Fanuc TP program (LS listing): hs0301h80_2.ls

/PROG  hs0301h80_2
/ATTR
COMMENT	= "19-03-01 11:47:14";
PROG_SIZE	= 0;
DEFAULT_GROUP	= 1, *, *, *, *;
/APPL
    ARC Welding Equipment: 1, *, *, *, *;
/MN
   1:  CALL HOME_ALL;
   1:  UFRAME_NUM = 1;
   1:  UTOOL_NUM = 3;
   1:  COL GUARD ADJUST 150;
   1:  PR[91] = PR[90];
   1:  PR[91,1] = PR[90,1] + -0.666;
   1:  PR[91,2] = PR[90,2] + 15.331;
   1:  PR[91,3] = PR[90,3] + 35.075;
   1:  PR[92] = PR[91];
   1:  PR[92,3] = PR[92,3] + 50;
   1:J PR[92] 10% FINE;
   1:L PR[91] R[100]mm/sec CNT100;
   1:  CALL LASER_DRAHT_START;
   1:  PR[91,1] = PR[90,1] + -0.927;
   1:  PR[91,2] = PR[90,2] + 15.462;
   1:L PR[91] R[100]mm/sec CNT100;
   1:  PR[91,1] = PR[90,1] + -1.615;
   1:  PR[91,2] = PR[90,2] + 15.721;
   1:L PR[91] R[100]mm/sec CNT100;
   1:  PR[91,1] = PR[90,1] + -2.354;
   1:  PR[91,2] = PR[90,2] + 16.306;
   1:L PR[91] R[100]mm/sec CNT100;
   1:  PR[91,1] = PR[90,1] + -3.858;
   1:  PR[91,2] = PR[90,2] + 17.303;
   1:L PR[91] R[100]mm/sec CNT100;
   1:  PR[91,1] = PR[90,1] + -4.809;
   1:  PR[91,2] = PR[90,2] + 17.719;
   1:L PR[91] R[100]mm/sec CNT100;
   1:  PR[91,1] = PR[90,1] + -8.585;
   1:  PR[91,2] = PR[90,2] + 19.301;
   1:L PR[91] R[100]mm/sec CNT100;
   1:  PR[91,1] = PR[90,1] + -9.692;
   1:  PR[91,2] = PR[90,2] + 19.587;
   1:L PR[91] R[100]mm/sec CNT100;
   1:  PR[91,1] = PR[90,1] + -11.119;
   1:  PR[91,2] = PR[90,2] + 19.736;
   1:L PR[91] R[100]mm/sec CNT100;
   1:  PR[91,1] = PR[90,1] + -14.708;
   1:  PR[91,2] = PR[90,2] + 20.226;
   1:L PR[91] R[100]mm/sec CNT100;
   1:  PR[91,1] = PR[90,1] + -16.221;
   1:  PR[91,2] = PR[90,2] + 20.146;
   1:L PR[91] R[100]mm/sec CNT100;
   1:  PR[91,1] = PR[90,1] + -19.349;
   1:  PR[91,2] = PR[90,2] + 19.776;
   1:L PR[91] R[100]mm/sec CNT100;
   1:  PR[91,1] = PR[90,1] + -20.989;
   1:  PR[91,2] = PR[90,2] + 19.436;
   1:L PR[91] R[100]mm/sec CNT100;
   1:  PR[91,1] = PR[90,1] + -22.810;
   1:  PR[91,2] = PR[90,2] + 18.760;
   1:L PR[91] R[100]mm/sec CNT100;
   1:  PR[91,1] = PR[90,1] + -25.231;
   1:  PR[91,2] = PR[90,2] + 17.813;
   1:L PR[91] R[100]mm/sec CNT100;
   1:  PR[91,1] = PR[90,1] + -26.962;
   1:  PR[91,2] = PR[90,2] + 16.843;
   1:L PR[91] R[100]mm/sec CNT100;
   1:  PR[91,1] = PR[90,1] + -28.774;
   1:  PR[91,2] = PR[90,2] + 15.433;
   1:L PR[91] R[100]mm/sec CNT100;
   1:  PR[91,1] = PR[90,1] + -30.430;
   1:  PR[91,2] = PR[90,2] + 14.227;
   1:L PR[91] R[100]mm/sec CNT100;
   1:  PR[91,1] = PR[90,1] + -31.950;
   1:  PR[91,2] = PR[90,2] + 12.586;
   1:L PR[91] R[100]mm/sec CNT100;
   1:  PR[91,1] = PR[90,1] + -33.021;
   1:  PR[91,2] = PR[90,2] + 11.255;
   1:L PR[91] R[100]mm/sec CNT100;
   1:  PR[91,1] = PR[90,1] + -34.310;
   1:  PR[91,2] = PR[90,2] + 9.296;
   1:L PR[91] R[100]mm/sec CNT100;
   1:  PR[91,1] = PR[90,1] + -35.922;
   1:  PR[91,2] = PR[90,2] + 5.672;
   1:L PR[91] R[100]mm/sec CNT100;
   1:  PR[91,1] = PR[90,1] + -36.506;
   1:  PR[91,2] = PR[90,2] + 3.415;
   1:L PR[91] R[100]mm/sec CNT100;
   1:  PR[91,1] = PR[90,1] + -36.709;
   1:  PR[91,2] = PR[90,2] + 0.880;
   1:L PR[91] R[100]mm/sec CNT100;
   1:  PR[91,1] = PR[90,1] + -36.880;
   1:  PR[91,2] = PR[90,2] + -0.354;
   1:L PR[91] R[100]mm/sec CNT100;
   1:  PR[91,1] = PR[90,1] + -36.688;
   1:  PR[91,2] = PR[90,2] + -2.767;
   1:L PR[91] R[100]mm/sec CNT100;
   1:  PR[91,1] = PR[90,1] + -36.517;
   1:  PR[91,2] = PR[90,2] + -3.999;
   1:L PR[91] R[100]mm/sec CNT100;
   1:  PR[91,1] = PR[90,1] + -35.922;
   1:  PR[91,2] = PR[90,2] + -6.296;
   1:L PR[91] R[100]mm/sec CNT100;
   1:  PR[91,1] = PR[90,1] + -34.892;
   1:  PR[91,2] = PR[90,2] + -8.592;
   1:L PR[91] R[100]mm/sec CNT100;
   1:  PR[91,1] = PR[90,1] + -34.306;
   1:  PR[91,2] = PR[90,2] + -9.927;
   1:L PR[91] R[100]mm/sec CNT100;
   1:  PR[91,1] = PR[90,1] + -33.019;
   1:  PR[91,2] = PR[90,2] + -11.883;
   1:L PR[91] R[100]mm/sec CNT100;
   1:  PR[91,1] = PR[90,1] + -31.945;
   1:  PR[91,2] = PR[90,2] + -13.214;
   1:L PR[91] R[100]mm/sec CNT100;
   1:  PR[91,1] = PR[90,1] + -30.408;
   1:  PR[91,2] = PR[90,2] + -14.874;
   1:L PR[91] R[100]mm/sec CNT100;
   1:  PR[91,1] = PR[90,1] + -28.736;
   1:  PR[91,2] = PR[90,2] + -16.183;
   1:L PR[91] R[100]mm/sec CNT100;
   1:  PR[91,1] = PR[90,1] + -26.973;
   1:  PR[91,2] = PR[90,2] + -17.461;
   1:L PR[91] R[100]mm/sec CNT100;
   1:  PR[91,1] = PR[90,1] + -25.232;
   1:  PR[91,2] = PR[90,2] + -18.437;
   1:L PR[91] R[100]mm/sec CNT100;
   1:  PR[91,1] = PR[90,1] + -23.475;
   1:  PR[91,2] = PR[90,2] + -19.085;
   1:L PR[91] R[100]mm/sec CNT100;
   1:  PR[91,1] = PR[90,1] + -20.959;
   1:  PR[91,2] = PR[90,2] + -20.067;
   1:L PR[91] R[100]mm/sec CNT100;
   1:  PR[91,1] = PR[90,1] + -19.331;
   1:  PR[91,2] = PR[90,2] + -20.404;
   1:L PR[91] R[100]mm/sec CNT100;
   1:  PR[91,1] = PR[90,1] + -16.196;
   1:  PR[91,2] = PR[90,2] + -20.770;
   1:L PR[91] R[100]mm/sec CNT100;
   1:  PR[91,1] = PR[90,1] + -14.656;
   1:  PR[91,2] = PR[90,2] + -20.851;
   1:L PR[91] R[100]mm/sec CNT100;
   1:  PR[91,1] = PR[90,1] + -13.288;
   1:  PR[91,2] = PR[90,2] + -20.713;
   1:L PR[91] R[100]mm/sec CNT100;
   1:  PR[91,1] = PR[90,1] + -9.682;
   1:  PR[91,2] = PR[90,2] + -20.208;
   1:L PR[91] R[100]mm/sec CNT100;
   1:  PR[91,1] = PR[90,1] + -8.557;
   1:  PR[91,2] = PR[90,2] + -19.917;
   1:L PR[91] R[100]mm/sec CNT100;
   1:  PR[91,1] = PR[90,1] + -3.731;
   1:  PR[91,2] = PR[90,2] + -17.847;
   1:L PR[91] R[100]mm/sec CNT100;
   1:  PR[91,1] = PR[90,1] + -3.017;
   1:  PR[91,2] = PR[90,2] + -17.391;
   1:L PR[91] R[100]mm/sec CNT100;
   1:  PR[91,1] = PR[90,1] + -1.910;
   1:  PR[91,2] = PR[90,2] + -16.593;
   1:L PR[91] R[100]mm/sec CNT100;
   1:  PR[91,1] = PR[90,1] + -1.659;
   1:  PR[91,2] = PR[90,2] + -16.373;
   1:L PR[91] R[100]mm/sec CNT100;
   1:  PR[91,1] = PR[90,1] + 0.008;
   1:  PR[91,2] = PR[90,2] + -15.711;
   1:L PR[91] R[100]mm/sec CNT100;
   1:  PR[91,1] = PR[90,1] + 0.793;
   1:  PR[91,2] = PR[90,2] + -16.025;
   1:L PR[91] R[100]mm/sec CNT100;
   1:  PR[91,1] = PR[90,1] + 1.694;
   1:  PR[91,2] = PR[90,2] + -16.187;
   1:L PR[91] R[100]mm/sec CNT100;
   1:  PR[91,1] = PR[90,1] + 2.030;
   1:  PR[91,2] = PR[90,2] + -16.568;
   1:L PR[91] R[100]mm/sec CNT100;
   1:  PR[91,1] = PR[90,1] + 2.042;
   1:  PR[91,2] = PR[90,2] + -16.578;
   1:L PR[91] R[100]mm/sec CNT100;
   1:  PR[91,1] = PR[90,1] + 2.791;
   1:  PR[91,2] = PR[90,2] + -17.107;
   1:L PR[91] R[100]mm/sec CNT100;
   1:  PR[91,1] = PR[90,1] + 3.899;
   1:  PR[91,2] = PR[90,2] + -17.854;
   1:L PR[91] R[100]mm/sec CNT100;
   1:  PR[91,1] = PR[90,1] + 8.708;
   1:  PR[91,2] = PR[90,2] + -19.914;
   1:L PR[91] R[100]mm/sec CNT100;
   1:  PR[91,1] = PR[90,1] + 9.812;
   1:  PR[91,2] = PR[90,2] + -20.200;
   1:L PR[91] R[100]mm/sec CNT100;
   1:  PR[91,1] = PR[90,1] + 11.237;
   1:  PR[91,2] = PR[90,2] + -20.349;
   1:L PR[91] R[100]mm/sec CNT100;
   1:  PR[91,1] = PR[90,1] + 14.834;
   1:  PR[91,2] = PR[90,2] + -20.850;
   1:L PR[91] R[100]mm/sec CNT100;
   1:  PR[91,1] = PR[90,1] + 16.338;
   1:  PR[91,2] = PR[90,2] + -20.771;
   1:L PR[91] R[100]mm/sec CNT100;
   1:  PR[91,1] = PR[90,1] + 19.474;
   1:  PR[91,2] = PR[90,2] + -20.406;
   1:L PR[91] R[100]mm/sec CNT100;
   1:  PR[91,1] = PR[90,1] + 21.112;
   1:  PR[91,2] = PR[90,2] + -20.067;
   1:L PR[91] R[100]mm/sec CNT100;
   1:  PR[91,1] = PR[90,1] + 22.936;
   1:  PR[91,2] = PR[90,2] + -19.393;
   1:L PR[91] R[100]mm/sec CNT100;
   1:  PR[91,1] = PR[90,1] + 25.366;
   1:  PR[91,2] = PR[90,2] + -18.448;
   1:L PR[91] R[100]mm/sec CNT100;
   1:  PR[91,1] = PR[90,1] + 27.089;
   1:  PR[91,2] = PR[90,2] + -17.488;
   1:L PR[91] R[100]mm/sec CNT100;
   1:  PR[91,1] = PR[90,1] + 28.887;
   1:  PR[91,2] = PR[90,2] + -16.095;
   1:L PR[91] R[100]mm/sec CNT100;
   1:  PR[91,1] = PR[90,1] + 30.549;
   1:  PR[91,2] = PR[90,2] + -14.888;
   1:L PR[91] R[100]mm/sec CNT100;
   1:  PR[91,1] = PR[90,1] + 32.072;
   1:  PR[91,2] = PR[90,2] + -13.246;
   1:L PR[91] R[100]mm/sec CNT100;
   1:  PR[91,1] = PR[90,1] + 33.148;
   1:  PR[91,2] = PR[90,2] + -11.909;
   1:L PR[91] R[100]mm/sec CNT100;
   1:  PR[91,1] = PR[90,1] + 34.457;
   1:  PR[91,2] = PR[90,2] + -9.931;
   1:L PR[91] R[100]mm/sec CNT100;
   1:  PR[91,1] = PR[90,1] + 35.518;
   1:  PR[91,2] = PR[90,2] + -7.595;
   1:L PR[91] R[100]mm/sec CNT100;
   1:  PR[91,1] = PR[90,1] + 36.065;
   1:  PR[91,2] = PR[90,2] + -6.353;
   1:L PR[91] R[100]mm/sec CNT100;
   1:  PR[91,1] = PR[90,1] + 36.652;
   1:  PR[91,2] = PR[90,2] + -4.119;
   1:L PR[91] R[100]mm/sec CNT100;
   1:  PR[91,1] = PR[90,1] + 36.866;
   1:  PR[91,2] = PR[90,2] + -1.508;
   1:L PR[91] R[100]mm/sec CNT100;
   1:  PR[91,1] = PR[90,1] + 37.037;
   1:  PR[91,2] = PR[90,2] + -0.271;
   1:L PR[91] R[100]mm/sec CNT100;
   1:  PR[91,1] = PR[90,1] + 36.834;
   1:  PR[91,2] = PR[90,2] + 2.220;
   1:L PR[91] R[100]mm/sec CNT100;
   1:  PR[91,1] = PR[90,1] + 36.662;
   1:  PR[91,2] = PR[90,2] + 3.454;
   1:L PR[91] R[100]mm/sec CNT100;
   1:  PR[91,1] = PR[90,1] + 36.068;
   1:  PR[91,2] = PR[90,2] + 5.720;
   1:L PR[91] R[100]mm/sec CNT100;
   1:  PR[91,1] = PR[90,1] + 35.039;
   1:  PR[91,2] = PR[90,2] + 7.981;
   1:L PR[91] R[100]mm/sec CNT100;
   1:  PR[91,1] = PR[90,1] + 34.455;
   1:  PR[91,2] = PR[90,2] + 9.310;
   1:L PR[91] R[100]mm/sec CNT100;
   1:  PR[91,1] = PR[90,1] + 33.150;
   1:  PR[91,2] = PR[90,2] + 11.281;
   1:L PR[91] R[100]mm/sec CNT100;
   1:  PR[91,1] = PR[90,1] + 32.076;
   1:  PR[91,2] = PR[90,2] + 12.617;
   1:L PR[91] R[100]mm/sec CNT100;
   1:  PR[91,1] = PR[90,1] + 30.537;
   1:  PR[91,2] = PR[90,2] + 14.277;
   1:L PR[91] R[100]mm/sec CNT100;
   1:  PR[91,1] = PR[90,1] + 28.879;
   1:  PR[91,2] = PR[90,2] + 15.569;
   1:L PR[91] R[100]mm/sec CNT100;
   1:  PR[91,1] = PR[90,1] + 27.119;
   1:  PR[91,2] = PR[90,2] + 16.848;
   1:L PR[91] R[100]mm/sec CNT100;
   1:  PR[91,1] = PR[90,1] + 25.389;
   1:  PR[91,2] = PR[90,2] + 17.812;
   1:L PR[91] R[100]mm/sec CNT100;
   1:  PR[91,1] = PR[90,1] + 23.629;
   1:  PR[91,2] = PR[90,2] + 18.459;
   1:L PR[91] R[100]mm/sec CNT100;
   1:  PR[91,1] = PR[90,1] + 21.116;
   1:  PR[91,2] = PR[90,2] + 19.442;
   1:L PR[91] R[100]mm/sec CNT100;
   1:  PR[91,1] = PR[90,1] + 19.492;
   1:  PR[91,2] = PR[90,2] + 19.778;
   1:L PR[91] R[100]mm/sec CNT100;
   1:  PR[91,1] = PR[90,1] + 16.363;
   1:  PR[91,2] = PR[90,2] + 20.148;
   1:L PR[91] R[100]mm/sec CNT100;
   1:  PR[91,1] = PR[90,1] + 14.834;
   1:  PR[91,2] = PR[90,2] + 20.227;
   1:L PR[91] R[100]mm/sec CNT100;
   1:  PR[91,1] = PR[90,1] + 13.468;
   1:  PR[91,2] = PR[90,2] + 20.089;
   1:L PR[91] R[100]mm/sec CNT100;
   1:  PR[91,1] = PR[90,1] + 9.868;
   1:  PR[91,2] = PR[90,2] + 19.591;
   1:L PR[91] R[100]mm/sec CNT100;
   1:  PR[91,1] = PR[90,1] + 8.747;
   1:  PR[91,2] = PR[90,2] + 19.300;
   1:L PR[91] R[100]mm/sec CNT100;
   1:  PR[91,1] = PR[90,1] + 7.722;
   1:  PR[91,2] = PR[90,2] + 18.852;
   1:L PR[91] R[100]mm/sec CNT100;
   1:  PR[91,1] = PR[90,1] + 3.989;
   1:  PR[91,2] = PR[90,2] + 17.292;
   1:L PR[91] R[100]mm/sec CNT100;
   1:  PR[91,1] = PR[90,1] + 3.235;
   1:  PR[91,2] = PR[90,2] + 16.810;
   1:L PR[91] R[100]mm/sec CNT100;
   1:  PR[91,1] = PR[90,1] + 2.521;
   1:  PR[91,2] = PR[90,2] + 16.318;
   1:L PR[91] R[100]mm/sec CNT100;
   1:  PR[91,1] = PR[90,1] + 2.001;
   1:  PR[91,2] = PR[90,2] + 15.906;
   1:L PR[91] R[100]mm/sec CNT100;
   1:  PR[91,1] = PR[90,1] + 1.619;
   1:  PR[91,2] = PR[90,2] + 15.536;
   1:L PR[91] R[100]mm/sec CNT100;
   1:  PR[91,1] = PR[90,1] + 0.760;
   1:  PR[91,2] = PR[90,2] + 15.389;
   1:L PR[91] R[100]mm/sec CNT100;
   1:  PR[91,1] = PR[90,1] + 0.087;
   1:  PR[91,2] = PR[90,2] + 15.117;
   1:L PR[91] R[100]mm/sec CNT100;
   1:  PR[91] = PR[90];
   1:  PR[91,1] = PR[90,1] + -0.722;
   1:  PR[91,2] = PR[90,2] + 15.588;
   1:  PR[91,3] = PR[90,3] + 35.685;
   1:L PR[91] R[100]mm/sec CNT100;
   1:  PR[91,1] = PR[90,1] + -1.091;
   1:  PR[91,2] = PR[90,2] + 15.774;
   1:L PR[91] R[100]mm/sec CNT100;
   1:  PR[91,1] = PR[90,1] + -1.597;
   1:  PR[91,2] = PR[90,2] + 15.965;
   1:L PR[91] R[100]mm/sec CNT100;
   1:  PR[91,1] = PR[90,1] + -2.135;
   1:  PR[91,2] = PR[90,2] + 16.391;
   1:L PR[91] R[100]mm/sec CNT100;
   1:  PR[91,1] = PR[90,1] + -3.572;
   1:  PR[91,2] = PR[90,2] + 17.346;
   1:L PR[91] R[100]mm/sec CNT100;
   1:  PR[91,1] = PR[90,1] + -4.394;
   1:  PR[91,2] = PR[90,2] + 17.706;
   1:L PR[91] R[100]mm/sec CNT100;
   1:  PR[91,1] = PR[90,1] + -8.389;
   1:  PR[91,2] = PR[90,2] + 19.380;
   1:L PR[91] R[100]mm/sec CNT100;
   1:  PR[91,1] = PR[90,1] + -9.367;
   1:  PR[91,2] = PR[90,2] + 19.633;
   1:L PR[91] R[100]mm/sec CNT100;
   1:  PR[91,1] = PR[90,1] + -10.645;
   1:  PR[91,2] = PR[90,2] + 19.766;
   1:L PR[91] R[100]mm/sec CNT100;
   1:  PR[91,1] = PR[90,1] + -14.484;
   1:  PR[91,2] = PR[90,2] + 20.290;
   1:L PR[91] R[100]mm/sec CNT100;
   1:  PR[91,1] = PR[90,1] + -15.854;
   1:  PR[91,2] = PR[90,2] + 20.217;
   1:L PR[91] R[100]mm/sec CNT100;
   1:  PR[91,1] = PR[90,1] + -19.224;
   1:  PR[91,2] = PR[90,2] + 19.819;
   1:L PR[91] R[100]mm/sec CNT100;
   1:  PR[91,1] = PR[90,1] + -20.730;
   1:  PR[91,2] = PR[90,2] + 19.506;
   1:L PR[91] R[100]mm/sec CNT100;
   1:  PR[91,1] = PR[90,1] + -22.409;
   1:  PR[91,2] = PR[90,2] + 18.883;
   1:L PR[91] R[100]mm/sec CNT100;
   1:  PR[91,1] = PR[90,1] + -25.070;
   1:  PR[91,2] = PR[90,2] + 17.843;
   1:L PR[91] R[100]mm/sec CNT100;
   1:  PR[91,1] = PR[90,1] + -26.674;
   1:  PR[91,2] = PR[90,2] + 16.944;
   1:L PR[91] R[100]mm/sec CNT100;
   1:  PR[91,1] = PR[90,1] + -28.363;
   1:  PR[91,2] = PR[90,2] + 15.630;
   1:L PR[91] R[100]mm/sec CNT100;
   1:  PR[91,1] = PR[90,1] + -30.234;
   1:  PR[91,2] = PR[90,2] + 14.267;
   1:L PR[91] R[100]mm/sec CNT100;
   1:  PR[91,1] = PR[90,1] + -31.654;
   1:  PR[91,2] = PR[90,2] + 12.733;
   1:L PR[91] R[100]mm/sec CNT100;
   1:  PR[91,1] = PR[90,1] + -32.885;
   1:  PR[91,2] = PR[90,2] + 11.204;
   1:L PR[91] R[100]mm/sec CNT100;
   1:  PR[91,1] = PR[90,1] + -34.095;
   1:  PR[91,2] = PR[90,2] + 9.366;
   1:L PR[91] R[100]mm/sec CNT100;
   1:  PR[91,1] = PR[90,1] + -35.747;
   1:  PR[91,2] = PR[90,2] + 5.647;
   1:L PR[91] R[100]mm/sec CNT100;
   1:  PR[91,1] = PR[90,1] + -36.296;
   1:  PR[91,2] = PR[90,2] + 3.526;
   1:L PR[91] R[100]mm/sec CNT100;
   1:  PR[91,1] = PR[90,1] + -36.488;
   1:  PR[91,2] = PR[90,2] + 1.135;
   1:L PR[91] R[100]mm/sec CNT100;
   1:  PR[91,1] = PR[90,1] + -36.694;
   1:  PR[91,2] = PR[90,2] + -0.354;
   1:L PR[91] R[100]mm/sec CNT100;
   1:  PR[91,1] = PR[90,1] + -36.513;
   1:  PR[91,2] = PR[90,2] + -2.628;
   1:L PR[91] R[100]mm/sec CNT100;
   1:  PR[91,1] = PR[90,1] + -36.306;
   1:  PR[91,2] = PR[90,2] + -4.111;
   1:L PR[91] R[100]mm/sec CNT100;
   1:  PR[91,1] = PR[90,1] + -35.747;
   1:  PR[91,2] = PR[90,2] + -6.271;
   1:L PR[91] R[100]mm/sec CNT100;
   1:  PR[91,1] = PR[90,1] + -34.776;
   1:  PR[91,2] = PR[90,2] + -8.435;
   1:L PR[91] R[100]mm/sec CNT100;
   1:  PR[91,1] = PR[90,1] + -34.091;
   1:  PR[91,2] = PR[90,2] + -9.996;
   1:L PR[91] R[100]mm/sec CNT100;
   1:  PR[91,1] = PR[90,1] + -32.883;
   1:  PR[91,2] = PR[90,2] + -11.832;
   1:L PR[91] R[100]mm/sec CNT100;
   1:  PR[91,1] = PR[90,1] + -31.648;
   1:  PR[91,2] = PR[90,2] + -13.363;
   1:L PR[91] R[100]mm/sec CNT100;
   1:  PR[91,1] = PR[90,1] + -30.211;
   1:  PR[91,2] = PR[90,2] + -14.915;
   1:L PR[91] R[100]mm/sec CNT100;
   1:  PR[91,1] = PR[90,1] + -28.647;
   1:  PR[91,2] = PR[90,2] + -16.139;
   1:L PR[91] R[100]mm/sec CNT100;
   1:  PR[91,1] = PR[90,1] + -26.684;
   1:  PR[91,2] = PR[90,2] + -17.563;
   1:L PR[91] R[100]mm/sec CNT100;
   1:  PR[91,1] = PR[90,1] + -25.069;
   1:  PR[91,2] = PR[90,2] + -18.467;
   1:L PR[91] R[100]mm/sec CNT100;
   1:  PR[91,1] = PR[90,1] + -23.435;
   1:  PR[91,2] = PR[90,2] + -19.071;
   1:L PR[91] R[100]mm/sec CNT100;
   1:  PR[91,1] = PR[90,1] + -20.699;
   1:  PR[91,2] = PR[90,2] + -20.138;
   1:L PR[91] R[100]mm/sec CNT100;
   1:  PR[91,1] = PR[90,1] + -19.205;
   1:  PR[91,2] = PR[90,2] + -20.448;
   1:L PR[91] R[100]mm/sec CNT100;
   1:  PR[91,1] = PR[90,1] + -15.826;
   1:  PR[91,2] = PR[90,2] + -20.841;
   1:L PR[91] R[100]mm/sec CNT100;
   1:  PR[91,1] = PR[90,1] + -14.430;
   1:  PR[91,2] = PR[90,2] + -20.915;
   1:L PR[91] R[100]mm/sec CNT100;
   1:  PR[91,1] = PR[90,1] + -13.190;
   1:  PR[91,2] = PR[90,2] + -20.790;
   1:L PR[91] R[100]mm/sec CNT100;
   1:  PR[91,1] = PR[90,1] + -9.355;
   1:  PR[91,2] = PR[90,2] + -20.253;
   1:L PR[91] R[100]mm/sec CNT100;
   1:  PR[91,1] = PR[90,1] + -8.359;
   1:  PR[91,2] = PR[90,2] + -19.996;
   1:L PR[91] R[100]mm/sec CNT100;
   1:  PR[91,1] = PR[90,1] + -3.437;
   1:  PR[91,2] = PR[90,2] + -17.886;
   1:L PR[91] R[100]mm/sec CNT100;
   1:  PR[91,1] = PR[90,1] + -2.832;
   1:  PR[91,2] = PR[90,2] + -17.500;
   1:L PR[91] R[100]mm/sec CNT100;
   1:  PR[91,1] = PR[90,1] + -1.582;
   1:  PR[91,2] = PR[90,2] + -16.598;
   1:L PR[91] R[100]mm/sec CNT100;
   1:  PR[91,1] = PR[90,1] + 0.021;
   1:  PR[91,2] = PR[90,2] + -15.944;
   1:L PR[91] R[100]mm/sec CNT100;
   1:  PR[91,1] = PR[90,1] + 1.017;
   1:  PR[91,2] = PR[90,2] + -16.343;
   1:L PR[91] R[100]mm/sec CNT100;
   1:  PR[91,1] = PR[90,1] + 1.715;
   1:  PR[91,2] = PR[90,2] + -16.468;
   1:L PR[91] R[100]mm/sec CNT100;
   1:  PR[91,1] = PR[90,1] + 2.003;
   1:  PR[91,2] = PR[90,2] + -16.795;
   1:L PR[91] R[100]mm/sec CNT100;
   1:  PR[91,1] = PR[90,1] + 2.436;
   1:  PR[91,2] = PR[90,2] + -17.104;
   1:L PR[91] R[100]mm/sec CNT100;
   1:  PR[91,1] = PR[90,1] + 3.606;
   1:  PR[91,2] = PR[90,2] + -17.893;
   1:L PR[91] R[100]mm/sec CNT100;
   1:  PR[91,1] = PR[90,1] + 8.511;
   1:  PR[91,2] = PR[90,2] + -19.992;
   1:L PR[91] R[100]mm/sec CNT100;
   1:  PR[91,1] = PR[90,1] + 9.485;
   1:  PR[91,2] = PR[90,2] + -20.245;
   1:L PR[91] R[100]mm/sec CNT100;
   1:  PR[91,1] = PR[90,1] + 10.761;
   1:  PR[91,2] = PR[90,2] + -20.379;
   1:L PR[91] R[100]mm/sec CNT100;
   1:  PR[91,1] = PR[90,1] + 14.609;
   1:  PR[91,2] = PR[90,2] + -20.914;
   1:L PR[91] R[100]mm/sec CNT100;
   1:  PR[91,1] = PR[90,1] + 15.970;
   1:  PR[91,2] = PR[90,2] + -20.843;
   1:L PR[91] R[100]mm/sec CNT100;
   1:  PR[91,1] = PR[90,1] + 19.349;
   1:  PR[91,2] = PR[90,2] + -20.449;
   1:L PR[91] R[100]mm/sec CNT100;
   1:  PR[91,1] = PR[90,1] + 20.853;
   1:  PR[91,2] = PR[90,2] + -20.138;
   1:L PR[91] R[100]mm/sec CNT100;
   1:  PR[91,1] = PR[90,1] + 22.535;
   1:  PR[91,2] = PR[90,2] + -19.517;
   1:L PR[91] R[100]mm/sec CNT100;
   1:  PR[91,1] = PR[90,1] + 25.204;
   1:  PR[91,2] = PR[90,2] + -18.479;
   1:L PR[91] R[100]mm/sec CNT100;
   1:  PR[91,1] = PR[90,1] + 26.802;
   1:  PR[91,2] = PR[90,2] + -17.589;
   1:L PR[91] R[100]mm/sec CNT100;
   1:  PR[91,1] = PR[90,1] + 28.476;
   1:  PR[91,2] = PR[90,2] + -16.291;
   1:L PR[91] R[100]mm/sec CNT100;
   1:  PR[91,1] = PR[90,1] + 30.354;
   1:  PR[91,2] = PR[90,2] + -14.927;
   1:L PR[91] R[100]mm/sec CNT100;
   1:  PR[91,1] = PR[90,1] + 31.777;
   1:  PR[91,2] = PR[90,2] + -13.392;
   1:L PR[91] R[100]mm/sec CNT100;
   1:  PR[91,1] = PR[90,1] + 33.014;
   1:  PR[91,2] = PR[90,2] + -11.856;
   1:L PR[91] R[100]mm/sec CNT100;
   1:  PR[91,1] = PR[90,1] + 34.242;
   1:  PR[91,2] = PR[90,2] + -10.000;
   1:L PR[91] R[100]mm/sec CNT100;
   1:  PR[91,1] = PR[90,1] + 35.240;
   1:  PR[91,2] = PR[90,2] + -7.803;
   1:L PR[91] R[100]mm/sec CNT100;
   1:  PR[91,1] = PR[90,1] + 35.891;
   1:  PR[91,2] = PR[90,2] + -6.326;
   1:L PR[91] R[100]mm/sec CNT100;
   1:  PR[91,1] = PR[90,1] + 36.442;
   1:  PR[91,2] = PR[90,2] + -4.227;
   1:L PR[91] R[100]mm/sec CNT100;
   1:  PR[91,1] = PR[90,1] + 36.644;
   1:  PR[91,2] = PR[90,2] + -1.764;
   1:L PR[91] R[100]mm/sec CNT100;
   1:  PR[91,1] = PR[90,1] + 36.851;
   1:  PR[91,2] = PR[90,2] + -0.271;
   1:L PR[91] R[100]mm/sec CNT100;
   1:  PR[91,1] = PR[90,1] + 36.659;
   1:  PR[91,2] = PR[90,2] + 2.076;
   1:L PR[91] R[100]mm/sec CNT100;
   1:  PR[91,1] = PR[90,1] + 36.453;
   1:  PR[91,2] = PR[90,2] + 3.562;
   1:L PR[91] R[100]mm/sec CNT100;
   1:  PR[91,1] = PR[90,1] + 35.894;
   1:  PR[91,2] = PR[90,2] + 5.692;
   1:L PR[91] R[100]mm/sec CNT100;
   1:  PR[91,1] = PR[90,1] + 34.924;
   1:  PR[91,2] = PR[90,2] + 7.824;
   1:L PR[91] R[100]mm/sec CNT100;
   1:  PR[91,1] = PR[90,1] + 34.240;
   1:  PR[91,2] = PR[90,2] + 9.379;
   1:L PR[91] R[100]mm/sec CNT100;
   1:  PR[91,1] = PR[90,1] + 33.016;
   1:  PR[91,2] = PR[90,2] + 11.228;
   1:L PR[91] R[100]mm/sec CNT100;
   1:  PR[91,1] = PR[90,1] + 31.782;
   1:  PR[91,2] = PR[90,2] + 12.763;
   1:L PR[91] R[100]mm/sec CNT100;
   1:  PR[91,1] = PR[90,1] + 30.343;
   1:  PR[91,2] = PR[90,2] + 14.315;
   1:L PR[91] R[100]mm/sec CNT100;
   1:  PR[91,1] = PR[90,1] + 28.792;
   1:  PR[91,2] = PR[90,2] + 15.524;
   1:L PR[91] R[100]mm/sec CNT100;
   1:  PR[91,1] = PR[90,1] + 26.833;
   1:  PR[91,2] = PR[90,2] + 16.947;
   1:L PR[91] R[100]mm/sec CNT100;
   1:  PR[91,1] = PR[90,1] + 25.228;
   1:  PR[91,2] = PR[90,2] + 17.841;
   1:L PR[91] R[100]mm/sec CNT100;
   1:  PR[91,1] = PR[90,1] + 23.590;
   1:  PR[91,2] = PR[90,2] + 18.443;
   1:L PR[91] R[100]mm/sec CNT100;
   1:  PR[91,1] = PR[90,1] + 20.859;
   1:  PR[91,2] = PR[90,2] + 19.512;
   1:L PR[91] R[100]mm/sec CNT100;
   1:  PR[91,1] = PR[90,1] + 19.367;
   1:  PR[91,2] = PR[90,2] + 19.821;
   1:L PR[91] R[100]mm/sec CNT100;
   1:  PR[91,1] = PR[90,1] + 15.997;
   1:  PR[91,2] = PR[90,2] + 20.219;
   1:L PR[91] R[100]mm/sec CNT100;
   1:  PR[91,1] = PR[90,1] + 14.610;
   1:  PR[91,2] = PR[90,2] + 20.291;
   1:L PR[91] R[100]mm/sec CNT100;
   1:  PR[91,1] = PR[90,1] + 13.371;
   1:  PR[91,2] = PR[90,2] + 20.166;
   1:L PR[91] R[100]mm/sec CNT100;
   1:  PR[91,1] = PR[90,1] + 9.543;
   1:  PR[91,2] = PR[90,2] + 19.636;
   1:L PR[91] R[100]mm/sec CNT100;
   1:  PR[91,1] = PR[90,1] + 8.551;
   1:  PR[91,2] = PR[90,2] + 19.379;
   1:L PR[91] R[100]mm/sec CNT100;
   1:  PR[91,1] = PR[90,1] + 7.637;
   1:  PR[91,2] = PR[90,2] + 18.979;
   1:L PR[91] R[100]mm/sec CNT100;
   1:  PR[91,1] = PR[90,1] + 3.702;
   1:  PR[91,2] = PR[90,2] + 17.335;
   1:L PR[91] R[100]mm/sec CNT100;
   1:  PR[91,1] = PR[90,1] + 3.052;
   1:  PR[91,2] = PR[90,2] + 16.920;
   1:L PR[91] R[100]mm/sec CNT100;
   1:  PR[91,1] = PR[90,1] + 2.311;
   1:  PR[91,2] = PR[90,2] + 16.408;
   1:L PR[91] R[100]mm/sec CNT100;
   1:  PR[91,1] = PR[90,1] + 1.574;
   1:  PR[91,2] = PR[90,2] + 15.805;
   1:L PR[91] R[100]mm/sec CNT100;
   1:  PR[91,1] = PR[90,1] + 0.969;
   1:  PR[91,2] = PR[90,2] + 15.702;
   1:L PR[91] R[100]mm/sec CNT100;
   1:  PR[91,1] = PR[90,1] + 0.107;
   1:  PR[91,2] = PR[90,2] + 15.353;
   1:L PR[91] R[100]mm/sec CNT100;
   1:  PR[91] = PR[90];
   1:  PR[91,1] = PR[90,1] + -0.777;
   1:  PR[91,2] = PR[90,2] + 15.846;
   1:  PR[91,3] = PR[90,3] + 36.295;
   1:L PR[91] R[100]mm/sec CNT100;
   1:  PR[91,1] = PR[90,1] + -1.255;
   1:  PR[91,2] = PR[90,2] + 16.087;
   1:L PR[91] R[100]mm/sec CNT100;
   1:  PR[91,1] = PR[90,1] + -1.580;
   1:  PR[91,2] = PR[90,2] + 16.209;
   1:L PR[91] R[100]mm/sec CNT100;
   1:  PR[91,1] = PR[90,1] + -1.917;
   1:  PR[91,2] = PR[90,2] + 16.476;
   1:L PR[91] R[100]mm/sec CNT100;
   1:  PR[91,1] = PR[90,1] + -3.286;
   1:  PR[91,2] = PR[90,2] + 17.390;
   1:L PR[91] R[100]mm/sec CNT100;
   1:  PR[91,1] = PR[90,1] + -3.979;
   1:  PR[91,2] = PR[90,2] + 17.693;
   1:L PR[91] R[100]mm/sec CNT100;
   1:  PR[91,1] = PR[90,1] + -8.193;
   1:  PR[91,2] = PR[90,2] + 19.459;
   1:L PR[91] R[100]mm/sec CNT100;
   1:  PR[91,1] = PR[90,1] + -9.042;
   1:  PR[91,2] = PR[90,2] + 19.678;
   1:L PR[91] R[100]mm/sec CNT100;
   1:  PR[91,1] = PR[90,1] + -10.171;
   1:  PR[91,2] = PR[90,2] + 19.796;
   1:L PR[91] R[100]mm/sec CNT100;
   1:  PR[91,1] = PR[90,1] + -14.260;
   1:  PR[91,2] = PR[90,2] + 20.354;
   1:L PR[91] R[100]mm/sec CNT100;
   1:  PR[91,1] = PR[90,1] + -15.487;
   1:  PR[91,2] = PR[90,2] + 20.289;
   1:L PR[91] R[100]mm/sec CNT100;
   1:  PR[91,1] = PR[90,1] + -19.099;
   1:  PR[91,2] = PR[90,2] + 19.862;
   1:L PR[91] R[100]mm/sec CNT100;
   1:  PR[91,1] = PR[90,1] + -20.472;
   1:  PR[91,2] = PR[90,2] + 19.577;
   1:L PR[91] R[100]mm/sec CNT100;
   1:  PR[91,1] = PR[90,1] + -22.008;
   1:  PR[91,2] = PR[90,2] + 19.007;
   1:L PR[91] R[100]mm/sec CNT100;
   1:  PR[91,1] = PR[90,1] + -24.908;
   1:  PR[91,2] = PR[90,2] + 17.873;
   1:L PR[91] R[100]mm/sec CNT100;
   1:  PR[91,1] = PR[90,1] + -26.386;
   1:  PR[91,2] = PR[90,2] + 17.045;
   1:L PR[91] R[100]mm/sec CNT100;
   1:  PR[91,1] = PR[90,1] + -27.951;
   1:  PR[91,2] = PR[90,2] + 15.827;
   1:L PR[91] R[100]mm/sec CNT100;
   1:  PR[91,1] = PR[90,1] + -30.038;
   1:  PR[91,2] = PR[90,2] + 14.307;
   1:L PR[91] R[100]mm/sec CNT100;
   1:  PR[91,1] = PR[90,1] + -31.358;
   1:  PR[91,2] = PR[90,2] + 12.881;
   1:L PR[91] R[100]mm/sec CNT100;
   1:  PR[91,1] = PR[90,1] + -32.750;
   1:  PR[91,2] = PR[90,2] + 11.153;
   1:L PR[91] R[100]mm/sec CNT100;
   1:  PR[91,1] = PR[90,1] + -33.880;
   1:  PR[91,2] = PR[90,2] + 9.435;
   1:L PR[91] R[100]mm/sec CNT100;
   1:  PR[91,1] = PR[90,1] + -35.572;
   1:  PR[91,2] = PR[90,2] + 5.622;
   1:L PR[91] R[100]mm/sec CNT100;
   1:  PR[91,1] = PR[90,1] + -36.086;
   1:  PR[91,2] = PR[90,2] + 3.637;
   1:L PR[91] R[100]mm/sec CNT100;
   1:  PR[91,1] = PR[90,1] + -36.266;
   1:  PR[91,2] = PR[90,2] + 1.389;
   1:L PR[91] R[100]mm/sec CNT100;
   1:  PR[91,1] = PR[90,1] + -36.508;
   1:  PR[91,2] = PR[90,2] + -0.354;
   1:L PR[91] R[100]mm/sec CNT100;
   1:  PR[91,1] = PR[90,1] + -36.338;
   1:  PR[91,2] = PR[90,2] + -2.488;
   1:L PR[91] R[100]mm/sec CNT100;
   1:  PR[91,1] = PR[90,1] + -36.096;
   1:  PR[91,2] = PR[90,2] + -4.222;
   1:L PR[91] R[100]mm/sec CNT100;
   1:  PR[91,1] = PR[90,1] + -35.572;
   1:  PR[91,2] = PR[90,2] + -6.245;
   1:L PR[91] R[100]mm/sec CNT100;
   1:  PR[91,1] = PR[90,1] + -34.660;
   1:  PR[91,2] = PR[90,2] + -8.278;
   1:L PR[91] R[100]mm/sec CNT100;
   1:  PR[91,1] = PR[90,1] + -33.876;
   1:  PR[91,2] = PR[90,2] + -10.066;
   1:L PR[91] R[100]mm/sec CNT100;
   1:  PR[91,1] = PR[90,1] + -32.747;
   1:  PR[91,2] = PR[90,2] + -11.782;
   1:L PR[91] R[100]mm/sec CNT100;
   1:  PR[91,1] = PR[90,1] + -31.352;
   1:  PR[91,2] = PR[90,2] + -13.511;
   1:L PR[91] R[100]mm/sec CNT100;
   1:  PR[91,1] = PR[90,1] + -30.014;
   1:  PR[91,2] = PR[90,2] + -14.956;
   1:L PR[91] R[100]mm/sec CNT100;
   1:  PR[91,1] = PR[90,1] + -28.558;
   1:  PR[91,2] = PR[90,2] + -16.096;
   1:L PR[91] R[100]mm/sec CNT100;
   1:  PR[91,1] = PR[90,1] + -26.395;
   1:  PR[91,2] = PR[90,2] + -17.664;
   1:L PR[91] R[100]mm/sec CNT100;
   1:  PR[91,1] = PR[90,1] + -24.907;
   1:  PR[91,2] = PR[90,2] + -18.498;
   1:L PR[91] R[100]mm/sec CNT100;
   1:  PR[91,1] = PR[90,1] + -23.395;
   1:  PR[91,2] = PR[90,2] + -19.056;
   1:L PR[91] R[100]mm/sec CNT100;
   1:  PR[91,1] = PR[90,1] + -20.439;
   1:  PR[91,2] = PR[90,2] + -20.209;
   1:L PR[91] R[100]mm/sec CNT100;
   1:  PR[91,1] = PR[90,1] + -19.078;
   1:  PR[91,2] = PR[90,2] + -20.491;
   1:L PR[91] R[100]mm/sec CNT100;
   1:  PR[91,1] = PR[90,1] + -15.457;
   1:  PR[91,2] = PR[90,2] + -20.913;
   1:L PR[91] R[100]mm/sec CNT100;
   1:  PR[91,1] = PR[90,1] + -14.204;
   1:  PR[91,2] = PR[90,2] + -20.979;
   1:L PR[91] R[100]mm/sec CNT100;
   1:  PR[91,1] = PR[90,1] + -13.091;
   1:  PR[91,2] = PR[90,2] + -20.867;
   1:L PR[91] R[100]mm/sec CNT100;
   1:  PR[91,1] = PR[90,1] + -9.028;
   1:  PR[91,2] = PR[90,2] + -20.298;
   1:L PR[91] R[100]mm/sec CNT100;
   1:  PR[91,1] = PR[90,1] + -8.161;
   1:  PR[91,2] = PR[90,2] + -20.074;
   1:L PR[91] R[100]mm/sec CNT100;
   1:  PR[91,1] = PR[90,1] + -3.144;
   1:  PR[91,2] = PR[90,2] + -17.925;
   1:L PR[91] R[100]mm/sec CNT100;
   1:  PR[91,1] = PR[90,1] + -2.648;
   1:  PR[91,2] = PR[90,2] + -17.608;
   1:L PR[91] R[100]mm/sec CNT100;
   1:  PR[91,1] = PR[90,1] + -1.505;
   1:  PR[91,2] = PR[90,2] + -16.784;
   1:L PR[91] R[100]mm/sec CNT100;
   1:  PR[91,1] = PR[90,1] + -1.236;
   1:  PR[91,2] = PR[90,2] + -16.705;
   1:L PR[91] R[100]mm/sec CNT100;
   1:  PR[91,1] = PR[90,1] + -0.025;
   1:  PR[91,2] = PR[90,2] + -16.206;
   1:L PR[91] R[100]mm/sec CNT100;
   1:  PR[91,1] = PR[90,1] + 0.729;
   1:  PR[91,2] = PR[90,2] + -16.437;
   1:L PR[91] R[100]mm/sec CNT100;
   1:  PR[91,1] = PR[90,1] + 0.941;
   1:  PR[91,2] = PR[90,2] + -16.548;
   1:L PR[91] R[100]mm/sec CNT100;
   1:  PR[91,1] = PR[90,1] + 1.231;
   1:  PR[91,2] = PR[90,2] + -16.659;
   1:L PR[91] R[100]mm/sec CNT100;
   1:  PR[91,1] = PR[90,1] + 1.580;
   1:  PR[91,2] = PR[90,2] + -16.721;
   1:L PR[91] R[100]mm/sec CNT100;
   1:  PR[91,1] = PR[90,1] + 2.095;
   1:  PR[91,2] = PR[90,2] + -17.110;
   1:L PR[91] R[100]mm/sec CNT100;
   1:  PR[91,1] = PR[90,1] + 3.312;
   1:  PR[91,2] = PR[90,2] + -17.932;
   1:L PR[91] R[100]mm/sec CNT100;
   1:  PR[91,1] = PR[90,1] + 8.313;
   1:  PR[91,2] = PR[90,2] + -20.071;
   1:L PR[91] R[100]mm/sec CNT100;
   1:  PR[91,1] = PR[90,1] + 9.158;
   1:  PR[91,2] = PR[90,2] + -20.290;
   1:L PR[91] R[100]mm/sec CNT100;
   1:  PR[91,1] = PR[90,1] + 10.286;
   1:  PR[91,2] = PR[90,2] + -20.408;
   1:L PR[91] R[100]mm/sec CNT100;
   1:  PR[91,1] = PR[90,1] + 14.383;
   1:  PR[91,2] = PR[90,2] + -20.978;
   1:L PR[91] R[100]mm/sec CNT100;
   1:  PR[91,1] = PR[90,1] + 15.602;
   1:  PR[91,2] = PR[90,2] + -20.914;
   1:L PR[91] R[100]mm/sec CNT100;
   1:  PR[91,1] = PR[90,1] + 19.223;
   1:  PR[91,2] = PR[90,2] + -20.492;
   1:L PR[91] R[100]mm/sec CNT100;
   1:  PR[91,1] = PR[90,1] + 20.594;
   1:  PR[91,2] = PR[90,2] + -20.209;
   1:L PR[91] R[100]mm/sec CNT100;
   1:  PR[91,1] = PR[90,1] + 22.133;
   1:  PR[91,2] = PR[90,2] + -19.640;
   1:L PR[91] R[100]mm/sec CNT100;
   1:  PR[91,1] = PR[90,1] + 25.043;
   1:  PR[91,2] = PR[90,2] + -18.509;
   1:L PR[91] R[100]mm/sec CNT100;
   1:  PR[91,1] = PR[90,1] + 26.514;
   1:  PR[91,2] = PR[90,2] + -17.689;
   1:L PR[91] R[100]mm/sec CNT100;
   1:  PR[91,1] = PR[90,1] + 28.065;
   1:  PR[91,2] = PR[90,2] + -16.487;
   1:L PR[91] R[100]mm/sec CNT100;
   1:  PR[91,1] = PR[90,1] + 30.159;
   1:  PR[91,2] = PR[90,2] + -14.966;
   1:L PR[91] R[100]mm/sec CNT100;
   1:  PR[91,1] = PR[90,1] + 31.482;
   1:  PR[91,2] = PR[90,2] + -13.539;
   1:L PR[91] R[100]mm/sec CNT100;
   1:  PR[91,1] = PR[90,1] + 32.880;
   1:  PR[91,2] = PR[90,2] + -11.804;
   1:L PR[91] R[100]mm/sec CNT100;
   1:  PR[91,1] = PR[90,1] + 34.028;
   1:  PR[91,2] = PR[90,2] + -10.068;
   1:L PR[91] R[100]mm/sec CNT100;
   1:  PR[91,1] = PR[90,1] + 34.962;
   1:  PR[91,2] = PR[90,2] + -8.011;
   1:L PR[91] R[100]mm/sec CNT100;
   1:  PR[91,1] = PR[90,1] + 35.717;
   1:  PR[91,2] = PR[90,2] + -6.299;
   1:L PR[91] R[100]mm/sec CNT100;
   1:  PR[91,1] = PR[90,1] + 36.232;
   1:  PR[91,2] = PR[90,2] + -4.335;
   1:L PR[91] R[100]mm/sec CNT100;
   1:  PR[91,1] = PR[90,1] + 36.422;
   1:  PR[91,2] = PR[90,2] + -2.020;
   1:L PR[91] R[100]mm/sec CNT100;
   1:  PR[91,1] = PR[90,1] + 36.664;
   1:  PR[91,2] = PR[90,2] + -0.271;
   1:L PR[91] R[100]mm/sec CNT100;
   1:  PR[91,1] = PR[90,1] + 36.485;
   1:  PR[91,2] = PR[90,2] + 1.933;
   1:L PR[91] R[100]mm/sec CNT100;
   1:  PR[91,1] = PR[90,1] + 36.243;
   1:  PR[91,2] = PR[90,2] + 3.669;
   1:L PR[91] R[100]mm/sec CNT100;
   1:  PR[91,1] = PR[90,1] + 35.720;
   1:  PR[91,2] = PR[90,2] + 5.664;
   1:L PR[91] R[100]mm/sec CNT100;
   1:  PR[91,1] = PR[90,1] + 34.809;
   1:  PR[91,2] = PR[90,2] + 7.667;
   1:L PR[91] R[100]mm/sec CNT100;
   1:  PR[91,1] = PR[90,1] + 34.026;
   1:  PR[91,2] = PR[90,2] + 9.447;
   1:L PR[91] R[100]mm/sec CNT100;
   1:  PR[91,1] = PR[90,1] + 32.882;
   1:  PR[91,2] = PR[90,2] + 11.175;
   1:L PR[91] R[100]mm/sec CNT100;
   1:  PR[91,1] = PR[90,1] + 31.488;
   1:  PR[91,2] = PR[90,2] + 12.909;
   1:L PR[91] R[100]mm/sec CNT100;
   1:  PR[91,1] = PR[90,1] + 30.149;
   1:  PR[91,2] = PR[90,2] + 14.353;
   1:L PR[91] R[100]mm/sec CNT100;
   1:  PR[91,1] = PR[90,1] + 28.705;
   1:  PR[91,2] = PR[90,2] + 15.479;
   1:L PR[91] R[100]mm/sec CNT100;
   1:  PR[91,1] = PR[90,1] + 26.547;
   1:  PR[91,2] = PR[90,2] + 17.047;
   1:L PR[91] R[100]mm/sec CNT100;
   1:  PR[91,1] = PR[90,1] + 25.068;
   1:  PR[91,2] = PR[90,2] + 17.871;
   1:L PR[91] R[100]mm/sec CNT100;
   1:  PR[91,1] = PR[90,1] + 23.551;
   1:  PR[91,2] = PR[90,2] + 18.428;
   1:L PR[91] R[100]mm/sec CNT100;
   1:  PR[91,1] = PR[90,1] + 20.602;
   1:  PR[91,2] = PR[90,2] + 19.582;
   1:L PR[91] R[100]mm/sec CNT100;
   1:  PR[91,1] = PR[90,1] + 19.243;
   1:  PR[91,2] = PR[90,2] + 19.863;
   1:L PR[91] R[100]mm/sec CNT100;
   1:  PR[91,1] = PR[90,1] + 15.631;
   1:  PR[91,2] = PR[90,2] + 20.291;
   1:L PR[91] R[100]mm/sec CNT100;
   1:  PR[91,1] = PR[90,1] + 14.386;
   1:  PR[91,2] = PR[90,2] + 20.355;
   1:L PR[91] R[100]mm/sec CNT100;
   1:  PR[91,1] = PR[90,1] + 13.273;
   1:  PR[91,2] = PR[90,2] + 20.242;
   1:L PR[91] R[100]mm/sec CNT100;
   1:  PR[91,1] = PR[90,1] + 9.218;
   1:  PR[91,2] = PR[90,2] + 19.682;
   1:L PR[91] R[100]mm/sec CNT100;
   1:  PR[91,1] = PR[90,1] + 8.356;
   1:  PR[91,2] = PR[90,2] + 19.458;
   1:L PR[91] R[100]mm/sec CNT100;
   1:  PR[91,1] = PR[90,1] + 7.551;
   1:  PR[91,2] = PR[90,2] + 19.106;
   1:L PR[91] R[100]mm/sec CNT100;
   1:  PR[91,1] = PR[90,1] + 3.415;
   1:  PR[91,2] = PR[90,2] + 17.377;
   1:L PR[91] R[100]mm/sec CNT100;
   1:  PR[91,1] = PR[90,1] + 2.869;
   1:  PR[91,2] = PR[90,2] + 17.029;
   1:L PR[91] R[100]mm/sec CNT100;
   1:  PR[91,1] = PR[90,1] + 2.090;
   1:  PR[91,2] = PR[90,2] + 16.491;
   1:L PR[91] R[100]mm/sec CNT100;
   1:  PR[91,1] = PR[90,1] + 1.594;
   1:  PR[91,2] = PR[90,2] + 16.085;
   1:L PR[91] R[100]mm/sec CNT100;
   1:  PR[91,1] = PR[90,1] + 1.177;
   1:  PR[91,2] = PR[90,2] + 16.014;
   1:L PR[91] R[100]mm/sec CNT100;
   1:  PR[91,1] = PR[90,1] + 0.127;
   1:  PR[91,2] = PR[90,2] + 15.590;
   1:L PR[91] R[100]mm/sec CNT100;
   1:  PR[91] = PR[90];
   1:  PR[91,1] = PR[90,1] + -0.833;
   1:  PR[91,2] = PR[90,2] + 16.104;
   1:  PR[91,3] = PR[90,3] + 36.905;
   1:L PR[91] R[100]mm/sec CNT100;
   1:  PR[91,1] = PR[90,1] + -1.572;
   1:  PR[91,2] = PR[90,2] + 16.475;
   1:L PR[91] R[100]mm/sec CNT100;
   1:  PR[91,1] = PR[90,1] + -2.992;
   1:  PR[91,2] = PR[90,2] + 17.428;
   1:L PR[91] R[100]mm/sec CNT100;
   1:  PR[91,1] = PR[90,1] + -7.999;
   1:  PR[91,2] = PR[90,2] + 19.538;
   1:L PR[91] R[100]mm/sec CNT100;
   1:  PR[91,1] = PR[90,1] + -8.717;
   1:  PR[91,2] = PR[90,2] + 19.723;
   1:L PR[91] R[100]mm/sec CNT100;
   1:  PR[91,1] = PR[90,1] + -9.698;
   1:  PR[91,2] = PR[90,2] + 19.826;
   1:L PR[91] R[100]mm/sec CNT100;
   1:  PR[91,1] = PR[90,1] + -14.036;
   1:  PR[91,2] = PR[90,2] + 20.418;
   1:L PR[91] R[100]mm/sec CNT100;
   1:  PR[91,1] = PR[90,1] + -15.119;
   1:  PR[91,2] = PR[90,2] + 20.361;
   1:L PR[91] R[100]mm/sec CNT100;
   1:  PR[91,1] = PR[90,1] + -18.974;
   1:  PR[91,2] = PR[90,2] + 19.905;
   1:L PR[91] R[100]mm/sec CNT100;
   1:  PR[91,1] = PR[90,1] + -20.214;
   1:  PR[91,2] = PR[90,2] + 19.648;
   1:L PR[91] R[100]mm/sec CNT100;
   1:  PR[91,1] = PR[90,1] + -21.607;
   1:  PR[91,2] = PR[90,2] + 19.131;
   1:L PR[91] R[100]mm/sec CNT100;
   1:  PR[91,1] = PR[90,1] + -24.747;
   1:  PR[91,2] = PR[90,2] + 17.903;
   1:L PR[91] R[100]mm/sec CNT100;
   1:  PR[91,1] = PR[90,1] + -26.099;
   1:  PR[91,2] = PR[90,2] + 17.145;
   1:L PR[91] R[100]mm/sec CNT100;
   1:  PR[91,1] = PR[90,1] + -27.539;
   1:  PR[91,2] = PR[90,2] + 16.024;
   1:L PR[91] R[100]mm/sec CNT100;
   1:  PR[91,1] = PR[90,1] + -29.842;
   1:  PR[91,2] = PR[90,2] + 14.347;
   1:L PR[91] R[100]mm/sec CNT100;
   1:  PR[91,1] = PR[90,1] + -31.062;
   1:  PR[91,2] = PR[90,2] + 13.029;
   1:L PR[91] R[100]mm/sec CNT100;
   1:  PR[91,1] = PR[90,1] + -32.614;
   1:  PR[91,2] = PR[90,2] + 11.102;
   1:L PR[91] R[100]mm/sec CNT100;
   1:  PR[91,1] = PR[90,1] + -33.665;
   1:  PR[91,2] = PR[90,2] + 9.505;
   1:L PR[91] R[100]mm/sec CNT100;
   1:  PR[91,1] = PR[90,1] + -35.397;
   1:  PR[91,2] = PR[90,2] + 5.597;
   1:L PR[91] R[100]mm/sec CNT100;
   1:  PR[91,1] = PR[90,1] + -35.876;
   1:  PR[91,2] = PR[90,2] + 3.749;
   1:L PR[91] R[100]mm/sec CNT100;
   1:  PR[91,1] = PR[90,1] + -36.044;
   1:  PR[91,2] = PR[90,2] + 1.644;
   1:L PR[91] R[100]mm/sec CNT100;
   1:  PR[91,1] = PR[90,1] + -36.321;
   1:  PR[91,2] = PR[90,2] + -0.354;
   1:L PR[91] R[100]mm/sec CNT100;
   1:  PR[91,1] = PR[90,1] + -36.163;
   1:  PR[91,2] = PR[90,2] + -2.349;
   1:L PR[91] R[100]mm/sec CNT100;
   1:  PR[91,1] = PR[90,1] + -35.886;
   1:  PR[91,2] = PR[90,2] + -4.334;
   1:L PR[91] R[100]mm/sec CNT100;
   1:  PR[91,1] = PR[90,1] + -35.397;
   1:  PR[91,2] = PR[90,2] + -6.220;
   1:L PR[91] R[100]mm/sec CNT100;
   1:  PR[91,1] = PR[90,1] + -34.544;
   1:  PR[91,2] = PR[90,2] + -8.121;
   1:L PR[91] R[100]mm/sec CNT100;
   1:  PR[91,1] = PR[90,1] + -33.661;
   1:  PR[91,2] = PR[90,2] + -10.136;
   1:L PR[91] R[100]mm/sec CNT100;
   1:  PR[91,1] = PR[90,1] + -32.611;
   1:  PR[91,2] = PR[90,2] + -11.731;
   1:L PR[91] R[100]mm/sec CNT100;
   1:  PR[91,1] = PR[90,1] + -31.055;
   1:  PR[91,2] = PR[90,2] + -13.660;
   1:L PR[91] R[100]mm/sec CNT100;
   1:  PR[91,1] = PR[90,1] + -29.817;
   1:  PR[91,2] = PR[90,2] + -14.997;
   1:L PR[91] R[100]mm/sec CNT100;
   1:  PR[91,1] = PR[90,1] + -28.469;
   1:  PR[91,2] = PR[90,2] + -16.052;
   1:L PR[91] R[100]mm/sec CNT100;
   1:  PR[91,1] = PR[90,1] + -26.106;
   1:  PR[91,2] = PR[90,2] + -17.765;
   1:L PR[91] R[100]mm/sec CNT100;
   1:  PR[91,1] = PR[90,1] + -24.744;
   1:  PR[91,2] = PR[90,2] + -18.528;
   1:L PR[91] R[100]mm/sec CNT100;
   1:  PR[91,1] = PR[90,1] + -23.354;
   1:  PR[91,2] = PR[90,2] + -19.041;
   1:L PR[91] R[100]mm/sec CNT100;
   1:  PR[91,1] = PR[90,1] + -20.179;
   1:  PR[91,2] = PR[90,2] + -20.280;
   1:L PR[91] R[100]mm/sec CNT100;
   1:  PR[91,1] = PR[90,1] + -18.952;
   1:  PR[91,2] = PR[90,2] + -20.534;
   1:L PR[91] R[100]mm/sec CNT100;
   1:  PR[91,1] = PR[90,1] + -15.088;
   1:  PR[91,2] = PR[90,2] + -20.984;
   1:L PR[91] R[100]mm/sec CNT100;
   1:  PR[91,1] = PR[90,1] + -13.978;
   1:  PR[91,2] = PR[90,2] + -21.043;
   1:L PR[91] R[100]mm/sec CNT100;
   1:  PR[91,1] = PR[90,1] + -12.992;
   1:  PR[91,2] = PR[90,2] + -20.943;
   1:L PR[91] R[100]mm/sec CNT100;
   1:  PR[91,1] = PR[90,1] + -8.701;
   1:  PR[91,2] = PR[90,2] + -20.343;
   1:L PR[91] R[100]mm/sec CNT100;
   1:  PR[91,1] = PR[90,1] + -7.963;
   1:  PR[91,2] = PR[90,2] + -20.152;
   1:L PR[91] R[100]mm/sec CNT100;
   1:  PR[91,1] = PR[90,1] + -2.850;
   1:  PR[91,2] = PR[90,2] + -17.964;
   1:L PR[91] R[100]mm/sec CNT100;
   1:  PR[91,1] = PR[90,1] + -2.462;
   1:  PR[91,2] = PR[90,2] + -17.716;
   1:L PR[91] R[100]mm/sec CNT100;
   1:  PR[91,1] = PR[90,1] + -1.487;
   1:  PR[91,2] = PR[90,2] + -17.013;
   1:L PR[91] R[100]mm/sec CNT100;
   1:  PR[91,1] = PR[90,1] + -1.147;
   1:  PR[91,2] = PR[90,2] + -16.913;
   1:L PR[91] R[100]mm/sec CNT100;
   1:  PR[91,1] = PR[90,1] + -0.005;
   1:  PR[91,2] = PR[90,2] + -16.442;
   1:L PR[91] R[100]mm/sec CNT100;
   1:  PR[91,1] = PR[90,1] + 0.784;
   1:  PR[91,2] = PR[90,2] + -16.684;
   1:L PR[91] R[100]mm/sec CNT100;
   1:  PR[91,1] = PR[90,1] + 1.038;
   1:  PR[91,2] = PR[90,2] + -16.817;
   1:L PR[91] R[100]mm/sec CNT100;
   1:  PR[91,1] = PR[90,1] + 1.666;
   1:  PR[91,2] = PR[90,2] + -17.058;
   1:L PR[91] R[100]mm/sec CNT100;
   1:  PR[91,1] = PR[90,1] + 3.019;
   1:  PR[91,2] = PR[90,2] + -17.971;
   1:L PR[91] R[100]mm/sec CNT100;
   1:  PR[91,1] = PR[90,1] + 8.115;
   1:  PR[91,2] = PR[90,2] + -20.149;
   1:L PR[91] R[100]mm/sec CNT100;
   1:  PR[91,1] = PR[90,1] + 8.831;
   1:  PR[91,2] = PR[90,2] + -20.334;
   1:L PR[91] R[100]mm/sec CNT100;
   1:  PR[91,1] = PR[90,1] + 9.810;
   1:  PR[91,2] = PR[90,2] + -20.437;
   1:L PR[91] R[100]mm/sec CNT100;
   1:  PR[91,1] = PR[90,1] + 14.157;
   1:  PR[91,2] = PR[90,2] + -21.042;
   1:L PR[91] R[100]mm/sec CNT100;
   1:  PR[91,1] = PR[90,1] + 15.234;
   1:  PR[91,2] = PR[90,2] + -20.986;
   1:L PR[91] R[100]mm/sec CNT100;
   1:  PR[91,1] = PR[90,1] + 19.098;
   1:  PR[91,2] = PR[90,2] + -20.536;
   1:L PR[91] R[100]mm/sec CNT100;
   1:  PR[91,1] = PR[90,1] + 20.335;
   1:  PR[91,2] = PR[90,2] + -20.279;
   1:L PR[91] R[100]mm/sec CNT100;
   1:  PR[91,1] = PR[90,1] + 21.731;
   1:  PR[91,2] = PR[90,2] + -19.764;
   1:L PR[91] R[100]mm/sec CNT100;
   1:  PR[91,1] = PR[90,1] + 24.881;
   1:  PR[91,2] = PR[90,2] + -18.539;
   1:L PR[91] R[100]mm/sec CNT100;
   1:  PR[91,1] = PR[90,1] + 26.226;
   1:  PR[91,2] = PR[90,2] + -17.789;
   1:L PR[91] R[100]mm/sec CNT100;
   1:  PR[91,1] = PR[90,1] + 27.654;
   1:  PR[91,2] = PR[90,2] + -16.683;
   1:L PR[91] R[100]mm/sec CNT100;
   1:  PR[91,1] = PR[90,1] + 29.964;
   1:  PR[91,2] = PR[90,2] + -15.005;
   1:L PR[91] R[100]mm/sec CNT100;
   1:  PR[91,1] = PR[90,1] + 31.187;
   1:  PR[91,2] = PR[90,2] + -13.686;
   1:L PR[91] R[100]mm/sec CNT100;
   1:  PR[91,1] = PR[90,1] + 32.745;
   1:  PR[91,2] = PR[90,2] + -11.751;
   1:L PR[91] R[100]mm/sec CNT100;
   1:  PR[91,1] = PR[90,1] + 33.813;
   1:  PR[91,2] = PR[90,2] + -10.137;
   1:L PR[91] R[100]mm/sec CNT100;
   1:  PR[91,1] = PR[90,1] + 34.684;
   1:  PR[91,2] = PR[90,2] + -8.219;
   1:L PR[91] R[100]mm/sec CNT100;
   1:  PR[91,1] = PR[90,1] + 35.543;
   1:  PR[91,2] = PR[90,2] + -6.271;
   1:L PR[91] R[100]mm/sec CNT100;
   1:  PR[91,1] = PR[90,1] + 36.023;
   1:  PR[91,2] = PR[90,2] + -4.443;
   1:L PR[91] R[100]mm/sec CNT100;
   1:  PR[91,1] = PR[90,1] + 36.201;
   1:  PR[91,2] = PR[90,2] + -2.275;
   1:L PR[91] R[100]mm/sec CNT100;
   1:  PR[91,1] = PR[90,1] + 36.478;
   1:  PR[91,2] = PR[90,2] + -0.271;
   1:L PR[91] R[100]mm/sec CNT100;
   1:  PR[91,1] = PR[90,1] + 36.310;
   1:  PR[91,2] = PR[90,2] + 1.789;
   1:L PR[91] R[100]mm/sec CNT100;
   1:  PR[91,1] = PR[90,1] + 36.034;
   1:  PR[91,2] = PR[90,2] + 3.777;
   1:L PR[91] R[100]mm/sec CNT100;
   1:  PR[91,1] = PR[90,1] + 35.546;
   1:  PR[91,2] = PR[90,2] + 5.637;
   1:L PR[91] R[100]mm/sec CNT100;
   1:  PR[91,1] = PR[90,1] + 34.694;
   1:  PR[91,2] = PR[90,2] + 7.509;
   1:L PR[91] R[100]mm/sec CNT100;
   1:  PR[91,1] = PR[90,1] + 33.812;
   1:  PR[91,2] = PR[90,2] + 9.515;
   1:L PR[91] R[100]mm/sec CNT100;
   1:  PR[91,1] = PR[90,1] + 32.748;
   1:  PR[91,2] = PR[90,2] + 11.122;
   1:L PR[91] R[100]mm/sec CNT100;
   1:  PR[91,1] = PR[90,1] + 31.194;
   1:  PR[91,2] = PR[90,2] + 13.055;
   1:L PR[91] R[100]mm/sec CNT100;
   1:  PR[91,1] = PR[90,1] + 29.955;
   1:  PR[91,2] = PR[90,2] + 14.392;
   1:L PR[91] R[100]mm/sec CNT100;
   1:  PR[91,1] = PR[90,1] + 28.618;
   1:  PR[91,2] = PR[90,2] + 15.434;
   1:L PR[91] R[100]mm/sec CNT100;
   1:  PR[91,1] = PR[90,1] + 26.260;
   1:  PR[91,2] = PR[90,2] + 17.147;
   1:L PR[91] R[100]mm/sec CNT100;
   1:  PR[91,1] = PR[90,1] + 24.907;
   1:  PR[91,2] = PR[90,2] + 17.901;
   1:L PR[91] R[100]mm/sec CNT100;
   1:  PR[91,1] = PR[90,1] + 23.513;
   1:  PR[91,2] = PR[90,2] + 18.413;
   1:L PR[91] R[100]mm/sec CNT100;
   1:  PR[91,1] = PR[90,1] + 20.344;
   1:  PR[91,2] = PR[90,2] + 19.653;
   1:L PR[91] R[100]mm/sec CNT100;
   1:  PR[91,1] = PR[90,1] + 19.119;
   1:  PR[91,2] = PR[90,2] + 19.906;
   1:L PR[91] R[100]mm/sec CNT100;
   1:  PR[91,1] = PR[90,1] + 15.265;
   1:  PR[91,2] = PR[90,2] + 20.362;
   1:L PR[91] R[100]mm/sec CNT100;
   1:  PR[91,1] = PR[90,1] + 14.162;
   1:  PR[91,2] = PR[90,2] + 20.419;
   1:L PR[91] R[100]mm/sec CNT100;
   1:  PR[91,1] = PR[90,1] + 13.176;
   1:  PR[91,2] = PR[90,2] + 20.319;
   1:L PR[91] R[100]mm/sec CNT100;
   1:  PR[91,1] = PR[90,1] + 8.893;
   1:  PR[91,2] = PR[90,2] + 19.727;
   1:L PR[91] R[100]mm/sec CNT100;
   1:  PR[91,1] = PR[90,1] + 8.160;
   1:  PR[91,2] = PR[90,2] + 19.537;
   1:L PR[91] R[100]mm/sec CNT100;
   1:  PR[91,1] = PR[90,1] + 7.466;
   1:  PR[91,2] = PR[90,2] + 19.233;
   1:L PR[91] R[100]mm/sec CNT100;
   1:  PR[91,1] = PR[90,1] + 3.127;
   1:  PR[91,2] = PR[90,2] + 17.420;
   1:L PR[91] R[100]mm/sec CNT100;
   1:  PR[91,1] = PR[90,1] + 2.687;
   1:  PR[91,2] = PR[90,2] + 17.139;
   1:L PR[91] R[100]mm/sec CNT100;
   1:  PR[91,1] = PR[90,1] + 1.683;
   1:  PR[91,2] = PR[90,2] + 16.445;
   1:L PR[91] R[100]mm/sec CNT100;
   1:  PR[91,1] = PR[90,1] + 0.146;
   1:  PR[91,2] = PR[90,2] + 15.826;
   1:L PR[91] R[100]mm/sec CNT100;
   1:  PR[91] = PR[90];
   1:  PR[91,1] = PR[90,1] + -0.893;
   1:  PR[91,2] = PR[90,2] + 16.363;
   1:  PR[91,3] = PR[90,3] + 37.515;
   1:L PR[91] R[100]mm/sec CNT100;
   1:  PR[91,1] = PR[90,1] + -1.558;
   1:  PR[91,2] = PR[90,2] + 16.702;
   1:L PR[91] R[100]mm/sec CNT100;
   1:  PR[91,1] = PR[90,1] + -2.704;
   1:  PR[91,2] = PR[90,2] + 17.470;
   1:L PR[91] R[100]mm/sec CNT100;
   1:  PR[91,1] = PR[90,1] + -7.803;
   1:  PR[91,2] = PR[90,2] + 19.617;
   1:L PR[91] R[100]mm/sec CNT100;
   1:  PR[91,1] = PR[90,1] + -8.392;
   1:  PR[91,2] = PR[90,2] + 19.769;
   1:L PR[91] R[100]mm/sec CNT100;
   1:  PR[91,1] = PR[90,1] + -9.224;
   1:  PR[91,2] = PR[90,2] + 19.856;
   1:L PR[91] R[100]mm/sec CNT100;
   1:  PR[91,1] = PR[90,1] + -13.812;
   1:  PR[91,2] = PR[90,2] + 20.482;
   1:L PR[91] R[100]mm/sec CNT100;
   1:  PR[91,1] = PR[90,1] + -14.752;
   1:  PR[91,2] = PR[90,2] + 20.432;
   1:L PR[91] R[100]mm/sec CNT100;
   1:  PR[91,1] = PR[90,1] + -18.849;
   1:  PR[91,2] = PR[90,2] + 19.948;
   1:L PR[91] R[100]mm/sec CNT100;
   1:  PR[91,1] = PR[90,1] + -19.955;
   1:  PR[91,2] = PR[90,2] + 19.718;
   1:L PR[91] R[100]mm/sec CNT100;
   1:  PR[91,1] = PR[90,1] + -21.206;
   1:  PR[91,2] = PR[90,2] + 19.254;
   1:L PR[91] R[100]mm/sec CNT100;
   1:  PR[91,1] = PR[90,1] + -24.585;
   1:  PR[91,2] = PR[90,2] + 17.933;
   1:L PR[91] R[100]mm/sec CNT100;
   1:  PR[91,1] = PR[90,1] + -25.811;
   1:  PR[91,2] = PR[90,2] + 17.246;
   1:L PR[91] R[100]mm/sec CNT100;
   1:  PR[91,1] = PR[90,1] + -27.127;
   1:  PR[91,2] = PR[90,2] + 16.222;
   1:L PR[91] R[100]mm/sec CNT100;
   1:  PR[91,1] = PR[90,1] + -29.646;
   1:  PR[91,2] = PR[90,2] + 14.387;
   1:L PR[91] R[100]mm/sec CNT100;
   1:  PR[91,1] = PR[90,1] + -30.766;
   1:  PR[91,2] = PR[90,2] + 13.177;
   1:L PR[91] R[100]mm/sec CNT100;
   1:  PR[91,1] = PR[90,1] + -32.478;
   1:  PR[91,2] = PR[90,2] + 11.051;
   1:L PR[91] R[100]mm/sec CNT100;
   1:  PR[91,1] = PR[90,1] + -33.450;
   1:  PR[91,2] = PR[90,2] + 9.574;
   1:L PR[91] R[100]mm/sec CNT100;
   1:  PR[91,1] = PR[90,1] + -35.223;
   1:  PR[91,2] = PR[90,2] + 5.571;
   1:L PR[91] R[100]mm/sec CNT100;
   1:  PR[91,1] = PR[90,1] + -35.666;
   1:  PR[91,2] = PR[90,2] + 3.860;
   1:L PR[91] R[100]mm/sec CNT100;
   1:  PR[91,1] = PR[90,1] + -35.823;
   1:  PR[91,2] = PR[90,2] + 1.899;
   1:L PR[91] R[100]mm/sec CNT100;
   1:  PR[91,1] = PR[90,1] + -36.135;
   1:  PR[91,2] = PR[90,2] + -0.354;
   1:L PR[91] R[100]mm/sec CNT100;
   1:  PR[91,1] = PR[90,1] + -35.988;
   1:  PR[91,2] = PR[90,2] + -2.209;
   1:L PR[91] R[100]mm/sec CNT100;
   1:  PR[91,1] = PR[90,1] + -35.676;
   1:  PR[91,2] = PR[90,2] + -4.446;
   1:L PR[91] R[100]mm/sec CNT100;
   1:  PR[91,1] = PR[90,1] + -35.223;
   1:  PR[91,2] = PR[90,2] + -6.195;
   1:L PR[91] R[100]mm/sec CNT100;
   1:  PR[91,1] = PR[90,1] + -34.429;
   1:  PR[91,2] = PR[90,2] + -7.964;
   1:L PR[91] R[100]mm/sec CNT100;
   1:  PR[91,1] = PR[90,1] + -33.445;
   1:  PR[91,2] = PR[90,2] + -10.206;
   1:L PR[91] R[100]mm/sec CNT100;
   1:  PR[91,1] = PR[90,1] + -32.475;
   1:  PR[91,2] = PR[90,2] + -11.680;
   1:L PR[91] R[100]mm/sec CNT100;
   1:  PR[91,1] = PR[90,1] + -30.758;
   1:  PR[91,2] = PR[90,2] + -13.809;
   1:L PR[91] R[100]mm/sec CNT100;
   1:  PR[91,1] = PR[90,1] + -29.620;
   1:  PR[91,2] = PR[90,2] + -15.038;
   1:L PR[91] R[100]mm/sec CNT100;
   1:  PR[91,1] = PR[90,1] + -28.380;
   1:  PR[91,2] = PR[90,2] + -16.008;
   1:L PR[91] R[100]mm/sec CNT100;
   1:  PR[91,1] = PR[90,1] + -25.817;
   1:  PR[91,2] = PR[90,2] + -17.867;
   1:L PR[91] R[100]mm/sec CNT100;
   1:  PR[91,1] = PR[90,1] + -24.582;
   1:  PR[91,2] = PR[90,2] + -18.559;
   1:L PR[91] R[100]mm/sec CNT100;
   1:  PR[91,1] = PR[90,1] + -23.314;
   1:  PR[91,2] = PR[90,2] + -19.027;
   1:L PR[91] R[100]mm/sec CNT100;
   1:  PR[91,1] = PR[90,1] + -19.919;
   1:  PR[91,2] = PR[90,2] + -20.351;
   1:L PR[91] R[100]mm/sec CNT100;
   1:  PR[91,1] = PR[90,1] + -18.826;
   1:  PR[91,2] = PR[90,2] + -20.578;
   1:L PR[91] R[100]mm/sec CNT100;
   1:  PR[91,1] = PR[90,1] + -14.719;
   1:  PR[91,2] = PR[90,2] + -21.056;
   1:L PR[91] R[100]mm/sec CNT100;
   1:  PR[91,1] = PR[90,1] + -13.752;
   1:  PR[91,2] = PR[90,2] + -21.107;
   1:L PR[91] R[100]mm/sec CNT100;
   1:  PR[91,1] = PR[90,1] + -12.893;
   1:  PR[91,2] = PR[90,2] + -21.020;
   1:L PR[91] R[100]mm/sec CNT100;
   1:  PR[91,1] = PR[90,1] + -8.374;
   1:  PR[91,2] = PR[90,2] + -20.388;
   1:L PR[91] R[100]mm/sec CNT100;
   1:  PR[91,1] = PR[90,1] + -7.765;
   1:  PR[91,2] = PR[90,2] + -20.230;
   1:L PR[91] R[100]mm/sec CNT100;
   1:  PR[91,1] = PR[90,1] + -2.557;
   1:  PR[91,2] = PR[90,2] + -18.003;
   1:L PR[91] R[100]mm/sec CNT100;
   1:  PR[91,1] = PR[90,1] + -2.277;
   1:  PR[91,2] = PR[90,2] + -17.824;
   1:L PR[91] R[100]mm/sec CNT100;
   1:  PR[91,1] = PR[90,1] + -1.470;
   1:  PR[91,2] = PR[90,2] + -17.242;
   1:L PR[91] R[100]mm/sec CNT100;
   1:  PR[91,1] = PR[90,1] + -1.059;
   1:  PR[91,2] = PR[90,2] + -17.121;
   1:L PR[91] R[100]mm/sec CNT100;
   1:  PR[91,1] = PR[90,1] + 0.015;
   1:  PR[91,2] = PR[90,2] + -16.678;
   1:L PR[91] R[100]mm/sec CNT100;
   1:  PR[91,1] = PR[90,1] + 0.838;
   1:  PR[91,2] = PR[90,2] + -16.930;
   1:L PR[91] R[100]mm/sec CNT100;
   1:  PR[91,1] = PR[90,1] + 1.135;
   1:  PR[91,2] = PR[90,2] + -17.086;
   1:L PR[91] R[100]mm/sec CNT100;
   1:  PR[91,1] = PR[90,1] + 1.649;
   1:  PR[91,2] = PR[90,2] + -17.283;
   1:L PR[91] R[100]mm/sec CNT100;
   1:  PR[91,1] = PR[90,1] + 2.726;
   1:  PR[91,2] = PR[90,2] + -18.010;
   1:L PR[91] R[100]mm/sec CNT100;
   1:  PR[91,1] = PR[90,1] + 7.918;
   1:  PR[91,2] = PR[90,2] + -20.227;
   1:L PR[91] R[100]mm/sec CNT100;
   1:  PR[91,1] = PR[90,1] + 8.504;
   1:  PR[91,2] = PR[90,2] + -20.379;
   1:L PR[91] R[100]mm/sec CNT100;
   1:  PR[91,1] = PR[90,1] + 9.334;
   1:  PR[91,2] = PR[90,2] + -20.466;
   1:L PR[91] R[100]mm/sec CNT100;
   1:  PR[91,1] = PR[90,1] + 13.932;
   1:  PR[91,2] = PR[90,2] + -21.106;
   1:L PR[91] R[100]mm/sec CNT100;
   1:  PR[91,1] = PR[90,1] + 14.866;
   1:  PR[91,2] = PR[90,2] + -21.057;
   1:L PR[91] R[100]mm/sec CNT100;
   1:  PR[91,1] = PR[90,1] + 18.972;
   1:  PR[91,2] = PR[90,2] + -20.579;
   1:L PR[91] R[100]mm/sec CNT100;
   1:  PR[91,1] = PR[90,1] + 20.077;
   1:  PR[91,2] = PR[90,2] + -20.350;
   1:L PR[91] R[100]mm/sec CNT100;
   1:  PR[91,1] = PR[90,1] + 21.329;
   1:  PR[91,2] = PR[90,2] + -19.887;
   1:L PR[91] R[100]mm/sec CNT100;
   1:  PR[91,1] = PR[90,1] + 24.719;
   1:  PR[91,2] = PR[90,2] + -18.569;
   1:L PR[91] R[100]mm/sec CNT100;
   1:  PR[91,1] = PR[90,1] + 25.939;
   1:  PR[91,2] = PR[90,2] + -17.890;
   1:L PR[91] R[100]mm/sec CNT100;
   1:  PR[91,1] = PR[90,1] + 27.244;
   1:  PR[91,2] = PR[90,2] + -16.879;
   1:L PR[91] R[100]mm/sec CNT100;
   1:  PR[91,1] = PR[90,1] + 29.769;
   1:  PR[91,2] = PR[90,2] + -15.044;
   1:L PR[91] R[100]mm/sec CNT100;
   1:  PR[91,1] = PR[90,1] + 30.892;
   1:  PR[91,2] = PR[90,2] + -13.833;
   1:L PR[91] R[100]mm/sec CNT100;
   1:  PR[91,1] = PR[90,1] + 32.611;
   1:  PR[91,2] = PR[90,2] + -11.699;
   1:L PR[91] R[100]mm/sec CNT100;
   1:  PR[91,1] = PR[90,1] + 33.599;
   1:  PR[91,2] = PR[90,2] + -10.206;
   1:L PR[91] R[100]mm/sec CNT100;
   1:  PR[91,1] = PR[90,1] + 34.406;
   1:  PR[91,2] = PR[90,2] + -8.427;
   1:L PR[91] R[100]mm/sec CNT100;
   1:  PR[91,1] = PR[90,1] + 35.369;
   1:  PR[91,2] = PR[90,2] + -6.244;
   1:L PR[91] R[100]mm/sec CNT100;
   1:  PR[91,1] = PR[90,1] + 35.813;
   1:  PR[91,2] = PR[90,2] + -4.551;
   1:L PR[91] R[100]mm/sec CNT100;
   1:  PR[91,1] = PR[90,1] + 35.979;
   1:  PR[91,2] = PR[90,2] + -2.531;
   1:L PR[91] R[100]mm/sec CNT100;
   1:  PR[91,1] = PR[90,1] + 36.292;
   1:  PR[91,2] = PR[90,2] + -0.271;
   1:L PR[91] R[100]mm/sec CNT100;
   1:  PR[91,1] = PR[90,1] + 36.136;
   1:  PR[91,2] = PR[90,2] + 1.645;
   1:L PR[91] R[100]mm/sec CNT100;
   1:  PR[91,1] = PR[90,1] + 35.824;
   1:  PR[91,2] = PR[90,2] + 3.885;
   1:L PR[91] R[100]mm/sec CNT100;
   1:  PR[91,1] = PR[90,1] + 35.372;
   1:  PR[91,2] = PR[90,2] + 5.609;
   1:L PR[91] R[100]mm/sec CNT100;
   1:  PR[91,1] = PR[90,1] + 34.579;
   1:  PR[91,2] = PR[90,2] + 7.352;
   1:L PR[91] R[100]mm/sec CNT100;
   1:  PR[91,1] = PR[90,1] + 33.598;
   1:  PR[91,2] = PR[90,2] + 9.583;
   1:L PR[91] R[100]mm/sec CNT100;
   1:  PR[91,1] = PR[90,1] + 32.614;
   1:  PR[91,2] = PR[90,2] + 11.069;
   1:L PR[91] R[100]mm/sec CNT100;
   1:  PR[91,1] = PR[90,1] + 30.900;
   1:  PR[91,2] = PR[90,2] + 13.202;
   1:L PR[91] R[100]mm/sec CNT100;
   1:  PR[91,1] = PR[90,1] + 29.761;
   1:  PR[91,2] = PR[90,2] + 14.430;
   1:L PR[91] R[100]mm/sec CNT100;
   1:  PR[91,1] = PR[90,1] + 28.531;
   1:  PR[91,2] = PR[90,2] + 15.389;
   1:L PR[91] R[100]mm/sec CNT100;
   1:  PR[91,1] = PR[90,1] + 25.974;
   1:  PR[91,2] = PR[90,2] + 17.246;
   1:L PR[91] R[100]mm/sec CNT100;
   1:  PR[91,1] = PR[90,1] + 24.746;
   1:  PR[91,2] = PR[90,2] + 17.930;
   1:L PR[91] R[100]mm/sec CNT100;
   1:  PR[91,1] = PR[90,1] + 23.474;
   1:  PR[91,2] = PR[90,2] + 18.398;
   1:L PR[91] R[100]mm/sec CNT100;
   1:  PR[91,1] = PR[90,1] + 20.087;
   1:  PR[91,2] = PR[90,2] + 19.723;
   1:L PR[91] R[100]mm/sec CNT100;
   1:  PR[91,1] = PR[90,1] + 18.995;
   1:  PR[91,2] = PR[90,2] + 19.949;
   1:L PR[91] R[100]mm/sec CNT100;
   1:  PR[91,1] = PR[90,1] + 14.898;
   1:  PR[91,2] = PR[90,2] + 20.433;
   1:L PR[91] R[100]mm/sec CNT100;
   1:  PR[91,1] = PR[90,1] + 13.938;
   1:  PR[91,2] = PR[90,2] + 20.483;
   1:L PR[91] R[100]mm/sec CNT100;
   1:  PR[91,1] = PR[90,1] + 13.079;
   1:  PR[91,2] = PR[90,2] + 20.396;
   1:L PR[91] R[100]mm/sec CNT100;
   1:  PR[91,1] = PR[90,1] + 8.568;
   1:  PR[91,2] = PR[90,2] + 19.773;
   1:L PR[91] R[100]mm/sec CNT100;
   1:  PR[91,1] = PR[90,1] + 7.964;
   1:  PR[91,2] = PR[90,2] + 19.616;
   1:L PR[91] R[100]mm/sec CNT100;
   1:  PR[91,1] = PR[90,1] + 7.380;
   1:  PR[91,2] = PR[90,2] + 19.360;
   1:L PR[91] R[100]mm/sec CNT100;
   1:  PR[91,1] = PR[90,1] + 2.840;
   1:  PR[91,2] = PR[90,2] + 17.463;
   1:L PR[91] R[100]mm/sec CNT100;
   1:  PR[91,1] = PR[90,1] + 2.504;
   1:  PR[91,2] = PR[90,2] + 17.249;
   1:L PR[91] R[100]mm/sec CNT100;
   1:  PR[91,1] = PR[90,1] + 1.668;
   1:  PR[91,2] = PR[90,2] + 16.671;
   1:L PR[91] R[100]mm/sec CNT100;
   1:  PR[91,1] = PR[90,1] + 0.169;
   1:  PR[91,2] = PR[90,2] + 16.062;
   1:L PR[91] R[100]mm/sec CNT100;
   1:  PR[91] = PR[90];
   1:  PR[91,1] = PR[90,1] + -0.953;
   1:  PR[91,2] = PR[90,2] + 16.622;
   1:  PR[91,3] = PR[90,3] + 38.125;
   1:L PR[91] R[100]mm/sec CNT100;
   1:  PR[91,1] = PR[90,1] + -1.544;
   1:  PR[91,2] = PR[90,2] + 16.928;
   1:L PR[91] R[100]mm/sec CNT100;
   1:  PR[91,1] = PR[90,1] + -2.425;
   1:  PR[91,2] = PR[90,2] + 17.519;
   1:L PR[91] R[100]mm/sec CNT100;
   1:  PR[91,1] = PR[90,1] + -2.733;
   1:  PR[91,2] = PR[90,2] + 17.653;
   1:L PR[91] R[100]mm/sec CNT100;
   1:  PR[91,1] = PR[90,1] + -7.606;
   1:  PR[91,2] = PR[90,2] + 19.695;
   1:L PR[91] R[100]mm/sec CNT100;
   1:  PR[91,1] = PR[90,1] + -8.067;
   1:  PR[91,2] = PR[90,2] + 19.814;
   1:L PR[91] R[100]mm/sec CNT100;
   1:  PR[91,1] = PR[90,1] + -8.750;
   1:  PR[91,2] = PR[90,2] + 19.886;
   1:L PR[91] R[100]mm/sec CNT100;
   1:  PR[91,1] = PR[90,1] + -13.588;
   1:  PR[91,2] = PR[90,2] + 20.546;
   1:L PR[91] R[100]mm/sec CNT100;
   1:  PR[91,1] = PR[90,1] + -14.385;
   1:  PR[91,2] = PR[90,2] + 20.504;
   1:L PR[91] R[100]mm/sec CNT100;
   1:  PR[91,1] = PR[90,1] + -18.724;
   1:  PR[91,2] = PR[90,2] + 19.991;
   1:L PR[91] R[100]mm/sec CNT100;
   1:  PR[91,1] = PR[90,1] + -19.697;
   1:  PR[91,2] = PR[90,2] + 19.789;
   1:L PR[91] R[100]mm/sec CNT100;
   1:  PR[91,1] = PR[90,1] + -20.805;
   1:  PR[91,2] = PR[90,2] + 19.378;
   1:L PR[91] R[100]mm/sec CNT100;
   1:  PR[91,1] = PR[90,1] + -24.424;
   1:  PR[91,2] = PR[90,2] + 17.963;
   1:L PR[91] R[100]mm/sec CNT100;
   1:  PR[91,1] = PR[90,1] + -25.523;
   1:  PR[91,2] = PR[90,2] + 17.347;
   1:L PR[91] R[100]mm/sec CNT100;
   1:  PR[91,1] = PR[90,1] + -26.716;
   1:  PR[91,2] = PR[90,2] + 16.419;
   1:L PR[91] R[100]mm/sec CNT100;
   1:  PR[91,1] = PR[90,1] + -29.450;
   1:  PR[91,2] = PR[90,2] + 14.427;
   1:L PR[91] R[100]mm/sec CNT100;
   1:  PR[91,1] = PR[90,1] + -30.470;
   1:  PR[91,2] = PR[90,2] + 13.325;
   1:L PR[91] R[100]mm/sec CNT100;
   1:  PR[91,1] = PR[90,1] + -32.343;
   1:  PR[91,2] = PR[90,2] + 11.000;
   1:L PR[91] R[100]mm/sec CNT100;
   1:  PR[91,1] = PR[90,1] + -33.235;
   1:  PR[91,2] = PR[90,2] + 9.644;
   1:L PR[91] R[100]mm/sec CNT100;
   1:  PR[91,1] = PR[90,1] + -35.048;
   1:  PR[91,2] = PR[90,2] + 5.546;
   1:L PR[91] R[100]mm/sec CNT100;
   1:  PR[91,1] = PR[90,1] + -35.456;
   1:  PR[91,2] = PR[90,2] + 3.971;
   1:L PR[91] R[100]mm/sec CNT100;
   1:  PR[91,1] = PR[90,1] + -35.601;
   1:  PR[91,2] = PR[90,2] + 2.154;
   1:L PR[91] R[100]mm/sec CNT100;
   1:  PR[91,1] = PR[90,1] + -35.949;
   1:  PR[91,2] = PR[90,2] + -0.354;
   1:L PR[91] R[100]mm/sec CNT100;
   1:  PR[91,1] = PR[90,1] + -35.812;
   1:  PR[91,2] = PR[90,2] + -2.070;
   1:L PR[91] R[100]mm/sec CNT100;
   1:  PR[91,1] = PR[90,1] + -35.465;
   1:  PR[91,2] = PR[90,2] + -4.557;
   1:L PR[91] R[100]mm/sec CNT100;
   1:  PR[91,1] = PR[90,1] + -35.048;
   1:  PR[91,2] = PR[90,2] + -6.170;
   1:L PR[91] R[100]mm/sec CNT100;
   1:  PR[91,1] = PR[90,1] + -34.313;
   1:  PR[91,2] = PR[90,2] + -7.808;
   1:L PR[91] R[100]mm/sec CNT100;
   1:  PR[91,1] = PR[90,1] + -33.230;
   1:  PR[91,2] = PR[90,2] + -10.276;
   1:L PR[91] R[100]mm/sec CNT100;
   1:  PR[91,1] = PR[90,1] + -32.339;
   1:  PR[91,2] = PR[90,2] + -11.630;
   1:L PR[91] R[100]mm/sec CNT100;
   1:  PR[91,1] = PR[90,1] + -30.462;
   1:  PR[91,2] = PR[90,2] + -13.957;
   1:L PR[91] R[100]mm/sec CNT100;
   1:  PR[91,1] = PR[90,1] + -29.424;
   1:  PR[91,2] = PR[90,2] + -15.079;
   1:L PR[91] R[100]mm/sec CNT100;
   1:  PR[91,1] = PR[90,1] + -28.291;
   1:  PR[91,2] = PR[90,2] + -15.965;
   1:L PR[91] R[100]mm/sec CNT100;
   1:  PR[91,1] = PR[90,1] + -25.528;
   1:  PR[91,2] = PR[90,2] + -17.968;
   1:L PR[91] R[100]mm/sec CNT100;
   1:  PR[91,1] = PR[90,1] + -24.419;
   1:  PR[91,2] = PR[90,2] + -18.589;
   1:L PR[91] R[100]mm/sec CNT100;
   1:  PR[91,1] = PR[90,1] + -23.273;
   1:  PR[91,2] = PR[90,2] + -19.012;
   1:L PR[91] R[100]mm/sec CNT100;
   1:  PR[91,1] = PR[90,1] + -19.659;
   1:  PR[91,2] = PR[90,2] + -20.422;
   1:L PR[91] R[100]mm/sec CNT100;
   1:  PR[91,1] = PR[90,1] + -18.699;
   1:  PR[91,2] = PR[90,2] + -20.621;
   1:L PR[91] R[100]mm/sec CNT100;
   1:  PR[91,1] = PR[90,1] + -14.350;
   1:  PR[91,2] = PR[90,2] + -21.127;
   1:L PR[91] R[100]mm/sec CNT100;
   1:  PR[91,1] = PR[90,1] + -13.526;
   1:  PR[91,2] = PR[90,2] + -21.171;
   1:L PR[91] R[100]mm/sec CNT100;
   1:  PR[91,1] = PR[90,1] + -12.794;
   1:  PR[91,2] = PR[90,2] + -21.097;
   1:L PR[91] R[100]mm/sec CNT100;
   1:  PR[91,1] = PR[90,1] + -8.047;
   1:  PR[91,2] = PR[90,2] + -20.433;
   1:L PR[91] R[100]mm/sec CNT100;
   1:  PR[91,1] = PR[90,1] + -7.567;
   1:  PR[91,2] = PR[90,2] + -20.309;
   1:L PR[91] R[100]mm/sec CNT100;
   1:  PR[91,1] = PR[90,1] + -2.264;
   1:  PR[91,2] = PR[90,2] + -18.042;
   1:L PR[91] R[100]mm/sec CNT100;
   1:  PR[91,1] = PR[90,1] + -2.092;
   1:  PR[91,2] = PR[90,2] + -17.932;
   1:L PR[91] R[100]mm/sec CNT100;
   1:  PR[91,1] = PR[90,1] + -1.453;
   1:  PR[91,2] = PR[90,2] + -17.471;
   1:L PR[91] R[100]mm/sec CNT100;
   1:  PR[91,1] = PR[90,1] + -0.971;
   1:  PR[91,2] = PR[90,2] + -17.329;
   1:L PR[91] R[100]mm/sec CNT100;
   1:  PR[91,1] = PR[90,1] + 0.035;
   1:  PR[91,2] = PR[90,2] + -16.914;
   1:L PR[91] R[100]mm/sec CNT100;
   1:  PR[91,1] = PR[90,1] + 0.892;
   1:  PR[91,2] = PR[90,2] + -17.177;
   1:L PR[91] R[100]mm/sec CNT100;
   1:  PR[91,1] = PR[90,1] + 1.233;
   1:  PR[91,2] = PR[90,2] + -17.355;
   1:L PR[91] R[100]mm/sec CNT100;
   1:  PR[91,1] = PR[90,1] + 1.631;
   1:  PR[91,2] = PR[90,2] + -17.508;
   1:L PR[91] R[100]mm/sec CNT100;
   1:  PR[91,1] = PR[90,1] + 2.437;
   1:  PR[91,2] = PR[90,2] + -18.052;
   1:L PR[91] R[100]mm/sec CNT100;
   1:  PR[91,1] = PR[90,1] + 2.680;
   1:  PR[91,2] = PR[90,2] + -18.158;
   1:L PR[91] R[100]mm/sec CNT100;
   1:  PR[91,1] = PR[90,1] + 7.719;
   1:  PR[91,2] = PR[90,2] + -20.306;
   1:L PR[91] R[100]mm/sec CNT100;
   1:  PR[91,1] = PR[90,1] + 8.177;
   1:  PR[91,2] = PR[90,2] + -20.424;
   1:L PR[91] R[100]mm/sec CNT100;
   1:  PR[91,1] = PR[90,1] + 8.859;
   1:  PR[91,2] = PR[90,2] + -20.496;
   1:L PR[91] R[100]mm/sec CNT100;
   1:  PR[91,1] = PR[90,1] + 13.706;
   1:  PR[91,2] = PR[90,2] + -21.170;
   1:L PR[91] R[100]mm/sec CNT100;
   1:  PR[91,1] = PR[90,1] + 14.498;
   1:  PR[91,2] = PR[90,2] + -21.129;
   1:L PR[91] R[100]mm/sec CNT100;
   1:  PR[91,1] = PR[90,1] + 18.847;
   1:  PR[91,2] = PR[90,2] + -20.622;
   1:L PR[91] R[100]mm/sec CNT100;
   1:  PR[91,1] = PR[90,1] + 19.818;
   1:  PR[91,2] = PR[90,2] + -20.421;
   1:L PR[91] R[100]mm/sec CNT100;
   1:  PR[91,1] = PR[90,1] + 20.927;
   1:  PR[91,2] = PR[90,2] + -20.011;
   1:L PR[91] R[100]mm/sec CNT100;
   1:  PR[91,1] = PR[90,1] + 24.557;
   1:  PR[91,2] = PR[90,2] + -18.600;
   1:L PR[91] R[100]mm/sec CNT100;
   1:  PR[91,1] = PR[90,1] + 25.651;
   1:  PR[91,2] = PR[90,2] + -17.990;
   1:L PR[91] R[100]mm/sec CNT100;
   1:  PR[91,1] = PR[90,1] + 26.833;
   1:  PR[91,2] = PR[90,2] + -17.074;
   1:L PR[91] R[100]mm/sec CNT100;
   1:  PR[91,1] = PR[90,1] + 29.574;
   1:  PR[91,2] = PR[90,2] + -15.083;
   1:L PR[91] R[100]mm/sec CNT100;
   1:  PR[91,1] = PR[90,1] + 30.597;
   1:  PR[91,2] = PR[90,2] + -13.980;
   1:L PR[91] R[100]mm/sec CNT100;
   1:  PR[91,1] = PR[90,1] + 32.476;
   1:  PR[91,2] = PR[90,2] + -11.646;
   1:L PR[91] R[100]mm/sec CNT100;
   1:  PR[91,1] = PR[90,1] + 33.384;
   1:  PR[91,2] = PR[90,2] + -10.274;
   1:L PR[91] R[100]mm/sec CNT100;
   1:  PR[91,1] = PR[90,1] + 34.129;
   1:  PR[91,2] = PR[90,2] + -8.635;
   1:L PR[91] R[100]mm/sec CNT100;
   1:  PR[91,1] = PR[90,1] + 35.195;
   1:  PR[91,2] = PR[90,2] + -6.217;
   1:L PR[91] R[100]mm/sec CNT100;
   1:  PR[91,1] = PR[90,1] + 35.604;
   1:  PR[91,2] = PR[90,2] + -4.659;
   1:L PR[91] R[100]mm/sec CNT100;
   1:  PR[91,1] = PR[90,1] + 35.757;
   1:  PR[91,2] = PR[90,2] + -2.787;
   1:L PR[91] R[100]mm/sec CNT100;
   1:  PR[91,1] = PR[90,1] + 36.105;
   1:  PR[91,2] = PR[90,2] + -0.271;
   1:L PR[91] R[100]mm/sec CNT100;
   1:  PR[91,1] = PR[90,1] + 35.961;
   1:  PR[91,2] = PR[90,2] + 1.502;
   1:L PR[91] R[100]mm/sec CNT100;
   1:  PR[91,1] = PR[90,1] + 35.615;
   1:  PR[91,2] = PR[90,2] + 3.992;
   1:L PR[91] R[100]mm/sec CNT100;
   1:  PR[91,1] = PR[90,1] + 35.198;
   1:  PR[91,2] = PR[90,2] + 5.581;
   1:L PR[91] R[100]mm/sec CNT100;
   1:  PR[91,1] = PR[90,1] + 34.464;
   1:  PR[91,2] = PR[90,2] + 7.195;
   1:L PR[91] R[100]mm/sec CNT100;
   1:  PR[91,1] = PR[90,1] + 33.383;
   1:  PR[91,2] = PR[90,2] + 9.651;
   1:L PR[91] R[100]mm/sec CNT100;
   1:  PR[91,1] = PR[90,1] + 32.480;
   1:  PR[91,2] = PR[90,2] + 11.016;
   1:L PR[91] R[100]mm/sec CNT100;
   1:  PR[91,1] = PR[90,1] + 30.605;
   1:  PR[91,2] = PR[90,2] + 13.348;
   1:L PR[91] R[100]mm/sec CNT100;
   1:  PR[91,1] = PR[90,1] + 29.567;
   1:  PR[91,2] = PR[90,2] + 14.468;
   1:L PR[91] R[100]mm/sec CNT100;
   1:  PR[91,1] = PR[90,1] + 28.444;
   1:  PR[91,2] = PR[90,2] + 15.343;
   1:L PR[91] R[100]mm/sec CNT100;
   1:  PR[91,1] = PR[90,1] + 25.687;
   1:  PR[91,2] = PR[90,2] + 17.346;
   1:L PR[91] R[100]mm/sec CNT100;
   1:  PR[91,1] = PR[90,1] + 24.585;
   1:  PR[91,2] = PR[90,2] + 17.960;
   1:L PR[91] R[100]mm/sec CNT100;
   1:  PR[91,1] = PR[90,1] + 23.436;
   1:  PR[91,2] = PR[90,2] + 18.383;
   1:L PR[91] R[100]mm/sec CNT100;
   1:  PR[91,1] = PR[90,1] + 19.830;
   1:  PR[91,2] = PR[90,2] + 19.793;
   1:L PR[91] R[100]mm/sec CNT100;
   1:  PR[91,1] = PR[90,1] + 18.871;
   1:  PR[91,2] = PR[90,2] + 19.992;
   1:L PR[91] R[100]mm/sec CNT100;
   1:  PR[91,1] = PR[90,1] + 14.532;
   1:  PR[91,2] = PR[90,2] + 20.505;
   1:L PR[91] R[100]mm/sec CNT100;
   1:  PR[91,1] = PR[90,1] + 13.714;
   1:  PR[91,2] = PR[90,2] + 20.547;
   1:L PR[91] R[100]mm/sec CNT100;
   1:  PR[91,1] = PR[90,1] + 12.982;
   1:  PR[91,2] = PR[90,2] + 20.473;
   1:L PR[91] R[100]mm/sec CNT100;
   1:  PR[91,1] = PR[90,1] + 8.243;
   1:  PR[91,2] = PR[90,2] + 19.818;
   1:L PR[91] R[100]mm/sec CNT100;
   1:  PR[91,1] = PR[90,1] + 7.758;
   1:  PR[91,2] = PR[90,2] + 19.692;
   1:L PR[91] R[100]mm/sec CNT100;
   1:  PR[91,1] = PR[90,1] + 2.568;
   1:  PR[91,2] = PR[90,2] + 17.513;
   1:L PR[91] R[100]mm/sec CNT100;
   1:  PR[91,1] = PR[90,1] + 1.643;
   1:  PR[91,2] = PR[90,2] + 16.892;
   1:L PR[91] R[100]mm/sec CNT100;
   1:  PR[91,1] = PR[90,1] + 0.192;
   1:  PR[91,2] = PR[90,2] + 16.297;
   1:L PR[91] R[100]mm/sec CNT100;
   1:  PR[91] = PR[90];
   1:  PR[91,1] = PR[90,1] + -1.016;
   1:  PR[91,2] = PR[90,2] + 16.882;
   1:  PR[91,3] = PR[90,3] + 38.735;
   1:L PR[91] R[100]mm/sec CNT100;
   1:  PR[91,1] = PR[90,1] + -1.533;
   1:  PR[91,2] = PR[90,2] + 17.156;
   1:L PR[91] R[100]mm/sec CNT100;
   1:  PR[91,1] = PR[90,1] + -2.138;
   1:  PR[91,2] = PR[90,2] + 17.562;
   1:L PR[91] R[100]mm/sec CNT100;
   1:  PR[91,1] = PR[90,1] + -2.317;
   1:  PR[91,2] = PR[90,2] + 17.640;
   1:L PR[91] R[100]mm/sec CNT100;
   1:  PR[91,1] = PR[90,1] + -7.410;
   1:  PR[91,2] = PR[90,2] + 19.774;
   1:L PR[91] R[100]mm/sec CNT100;
   1:  PR[91,1] = PR[90,1] + -7.742;
   1:  PR[91,2] = PR[90,2] + 19.860;
   1:L PR[91] R[100]mm/sec CNT100;
   1:  PR[91,1] = PR[90,1] + -8.276;
   1:  PR[91,2] = PR[90,2] + 19.915;
   1:L PR[91] R[100]mm/sec CNT100;
   1:  PR[91,1] = PR[90,1] + -13.363;
   1:  PR[91,2] = PR[90,2] + 20.610;
   1:L PR[91] R[100]mm/sec CNT100;
   1:  PR[91,1] = PR[90,1] + -14.018;
   1:  PR[91,2] = PR[90,2] + 20.575;
   1:L PR[91] R[100]mm/sec CNT100;
   1:  PR[91,1] = PR[90,1] + -18.599;
   1:  PR[91,2] = PR[90,2] + 20.034;
   1:L PR[91] R[100]mm/sec CNT100;
   1:  PR[91,1] = PR[90,1] + -19.439;
   1:  PR[91,2] = PR[90,2] + 19.859;
   1:L PR[91] R[100]mm/sec CNT100;
   1:  PR[91,1] = PR[90,1] + -20.404;
   1:  PR[91,2] = PR[90,2] + 19.501;
   1:L PR[91] R[100]mm/sec CNT100;
   1:  PR[91,1] = PR[90,1] + -24.262;
   1:  PR[91,2] = PR[90,2] + 17.993;
   1:L PR[91] R[100]mm/sec CNT100;
   1:  PR[91,1] = PR[90,1] + -25.236;
   1:  PR[91,2] = PR[90,2] + 17.447;
   1:L PR[91] R[100]mm/sec CNT100;
   1:  PR[91,1] = PR[90,1] + -26.304;
   1:  PR[91,2] = PR[90,2] + 16.616;
   1:L PR[91] R[100]mm/sec CNT100;
   1:  PR[91,1] = PR[90,1] + -29.253;
   1:  PR[91,2] = PR[90,2] + 14.468;
   1:L PR[91] R[100]mm/sec CNT100;
   1:  PR[91,1] = PR[90,1] + -30.174;
   1:  PR[91,2] = PR[90,2] + 13.473;
   1:L PR[91] R[100]mm/sec CNT100;
   1:  PR[91,1] = PR[90,1] + -32.207;
   1:  PR[91,2] = PR[90,2] + 10.949;
   1:L PR[91] R[100]mm/sec CNT100;
   1:  PR[91,1] = PR[90,1] + -33.020;
   1:  PR[91,2] = PR[90,2] + 9.713;
   1:L PR[91] R[100]mm/sec CNT100;
   1:  PR[91,1] = PR[90,1] + -34.873;
   1:  PR[91,2] = PR[90,2] + 5.521;
   1:L PR[91] R[100]mm/sec CNT100;
   1:  PR[91,1] = PR[90,1] + -35.246;
   1:  PR[91,2] = PR[90,2] + 4.082;
   1:L PR[91] R[100]mm/sec CNT100;
   1:  PR[91,1] = PR[90,1] + -35.380;
   1:  PR[91,2] = PR[90,2] + 2.409;
   1:L PR[91] R[100]mm/sec CNT100;
   1:  PR[91,1] = PR[90,1] + -35.763;
   1:  PR[91,2] = PR[90,2] + -0.354;
   1:L PR[91] R[100]mm/sec CNT100;
   1:  PR[91,1] = PR[90,1] + -35.637;
   1:  PR[91,2] = PR[90,2] + -1.930;
   1:L PR[91] R[100]mm/sec CNT100;
   1:  PR[91,1] = PR[90,1] + -35.255;
   1:  PR[91,2] = PR[90,2] + -4.669;
   1:L PR[91] R[100]mm/sec CNT100;
   1:  PR[91,1] = PR[90,1] + -34.873;
   1:  PR[91,2] = PR[90,2] + -6.144;
   1:L PR[91] R[100]mm/sec CNT100;
   1:  PR[91,1] = PR[90,1] + -34.197;
   1:  PR[91,2] = PR[90,2] + -7.651;
   1:L PR[91] R[100]mm/sec CNT100;
   1:  PR[91,1] = PR[90,1] + -33.015;
   1:  PR[91,2] = PR[90,2] + -10.346;
   1:L PR[91] R[100]mm/sec CNT100;
   1:  PR[91,1] = PR[90,1] + -32.203;
   1:  PR[91,2] = PR[90,2] + -11.579;
   1:L PR[91] R[100]mm/sec CNT100;
   1:  PR[91,1] = PR[90,1] + -30.165;
   1:  PR[91,2] = PR[90,2] + -14.106;
   1:L PR[91] R[100]mm/sec CNT100;
   1:  PR[91,1] = PR[90,1] + -29.227;
   1:  PR[91,2] = PR[90,2] + -15.119;
   1:L PR[91] R[100]mm/sec CNT100;
   1:  PR[91,1] = PR[90,1] + -28.202;
   1:  PR[91,2] = PR[90,2] + -15.921;
   1:L PR[91] R[100]mm/sec CNT100;
   1:  PR[91,1] = PR[90,1] + -25.239;
   1:  PR[91,2] = PR[90,2] + -18.069;
   1:L PR[91] R[100]mm/sec CNT100;
   1:  PR[91,1] = PR[90,1] + -24.256;
   1:  PR[91,2] = PR[90,2] + -18.620;
   1:L PR[91] R[100]mm/sec CNT100;
   1:  PR[91,1] = PR[90,1] + -23.233;
   1:  PR[91,2] = PR[90,2] + -18.998;
   1:L PR[91] R[100]mm/sec CNT100;
   1:  PR[91,1] = PR[90,1] + -19.399;
   1:  PR[91,2] = PR[90,2] + -20.493;
   1:L PR[91] R[100]mm/sec CNT100;
   1:  PR[91,1] = PR[90,1] + -18.573;
   1:  PR[91,2] = PR[90,2] + -20.664;
   1:L PR[91] R[100]mm/sec CNT100;
   1:  PR[91,1] = PR[90,1] + -13.981;
   1:  PR[91,2] = PR[90,2] + -21.199;
   1:L PR[91] R[100]mm/sec CNT100;
   1:  PR[91,1] = PR[90,1] + -13.300;
   1:  PR[91,2] = PR[90,2] + -21.235;
   1:L PR[91] R[100]mm/sec CNT100;
   1:  PR[91,1] = PR[90,1] + -12.695;
   1:  PR[91,2] = PR[90,2] + -21.174;
   1:L PR[91] R[100]mm/sec CNT100;
   1:  PR[91,1] = PR[90,1] + -7.720;
   1:  PR[91,2] = PR[90,2] + -20.478;
   1:L PR[91] R[100]mm/sec CNT100;
   1:  PR[91,1] = PR[90,1] + -7.369;
   1:  PR[91,2] = PR[90,2] + -20.387;
   1:L PR[91] R[100]mm/sec CNT100;
   1:  PR[91,1] = PR[90,1] + -1.993;
   1:  PR[91,2] = PR[90,2] + -18.091;
   1:L PR[91] R[100]mm/sec CNT100;
   1:  PR[91,1] = PR[90,1] + -1.420;
   1:  PR[91,2] = PR[90,2] + -17.696;
   1:L PR[91] R[100]mm/sec CNT100;
   1:  PR[91,1] = PR[90,1] + -0.882;
   1:  PR[91,2] = PR[90,2] + -17.538;
   1:L PR[91] R[100]mm/sec CNT100;
   1:  PR[91,1] = PR[90,1] + 0.055;
   1:  PR[91,2] = PR[90,2] + -17.151;
   1:L PR[91] R[100]mm/sec CNT100;
   1:  PR[91,1] = PR[90,1] + 0.947;
   1:  PR[91,2] = PR[90,2] + -17.424;
   1:L PR[91] R[100]mm/sec CNT100;
   1:  PR[91,1] = PR[90,1] + 1.330;
   1:  PR[91,2] = PR[90,2] + -17.624;
   1:L PR[91] R[100]mm/sec CNT100;
   1:  PR[91,1] = PR[90,1] + 1.614;
   1:  PR[91,2] = PR[90,2] + -17.734;
   1:L PR[91] R[100]mm/sec CNT100;
   1:  PR[91,1] = PR[90,1] + 2.144;
   1:  PR[91,2] = PR[90,2] + -18.091;
   1:L PR[91] R[100]mm/sec CNT100;
   1:  PR[91,1] = PR[90,1] + 2.255;
   1:  PR[91,2] = PR[90,2] + -18.140;
   1:L PR[91] R[100]mm/sec CNT100;
   1:  PR[91,1] = PR[90,1] + 7.522;
   1:  PR[91,2] = PR[90,2] + -20.384;
   1:L PR[91] R[100]mm/sec CNT100;
   1:  PR[91,1] = PR[90,1] + 7.850;
   1:  PR[91,2] = PR[90,2] + -20.469;
   1:L PR[91] R[100]mm/sec CNT100;
   1:  PR[91,1] = PR[90,1] + 8.383;
   1:  PR[91,2] = PR[90,2] + -20.525;
   1:L PR[91] R[100]mm/sec CNT100;
   1:  PR[91,1] = PR[90,1] + 13.480;
   1:  PR[91,2] = PR[90,2] + -21.234;
   1:L PR[91] R[100]mm/sec CNT100;
   1:  PR[91,1] = PR[90,1] + 14.129;
   1:  PR[91,2] = PR[90,2] + -21.200;
   1:L PR[91] R[100]mm/sec CNT100;
   1:  PR[91,1] = PR[90,1] + 18.721;
   1:  PR[91,2] = PR[90,2] + -20.665;
   1:L PR[91] R[100]mm/sec CNT100;
   1:  PR[91,1] = PR[90,1] + 19.559;
   1:  PR[91,2] = PR[90,2] + -20.492;
   1:L PR[91] R[100]mm/sec CNT100;
   1:  PR[91,1] = PR[90,1] + 20.526;
   1:  PR[91,2] = PR[90,2] + -20.135;
   1:L PR[91] R[100]mm/sec CNT100;
   1:  PR[91,1] = PR[90,1] + 24.395;
   1:  PR[91,2] = PR[90,2] + -18.630;
   1:L PR[91] R[100]mm/sec CNT100;
   1:  PR[91,1] = PR[90,1] + 25.364;
   1:  PR[91,2] = PR[90,2] + -18.090;
   1:L PR[91] R[100]mm/sec CNT100;
   1:  PR[91,1] = PR[90,1] + 26.422;
   1:  PR[91,2] = PR[90,2] + -17.270;
   1:L PR[91] R[100]mm/sec CNT100;
   1:  PR[91,1] = PR[90,1] + 29.379;
   1:  PR[91,2] = PR[90,2] + -15.122;
   1:L PR[91] R[100]mm/sec CNT100;
   1:  PR[91,1] = PR[90,1] + 30.302;
   1:  PR[91,2] = PR[90,2] + -14.127;
   1:L PR[91] R[100]mm/sec CNT100;
   1:  PR[91,1] = PR[90,1] + 32.342;
   1:  PR[91,2] = PR[90,2] + -11.594;
   1:L PR[91] R[100]mm/sec CNT100;
   1:  PR[91,1] = PR[90,1] + 33.170;
   1:  PR[91,2] = PR[90,2] + -10.343;
   1:L PR[91] R[100]mm/sec CNT100;
   1:  PR[91,1] = PR[90,1] + 33.851;
   1:  PR[91,2] = PR[90,2] + -8.842;
   1:L PR[91] R[100]mm/sec CNT100;
   1:  PR[91,1] = PR[90,1] + 35.021;
   1:  PR[91,2] = PR[90,2] + -6.189;
   1:L PR[91] R[100]mm/sec CNT100;
   1:  PR[91,1] = PR[90,1] + 35.394;
   1:  PR[91,2] = PR[90,2] + -4.767;
   1:L PR[91] R[100]mm/sec CNT100;
   1:  PR[91,1] = PR[90,1] + 35.535;
   1:  PR[91,2] = PR[90,2] + -3.043;
   1:L PR[91] R[100]mm/sec CNT100;
   1:  PR[91,1] = PR[90,1] + 35.919;
   1:  PR[91,2] = PR[90,2] + -0.271;
   1:L PR[91] R[100]mm/sec CNT100;
   1:  PR[91,1] = PR[90,1] + 35.786;
   1:  PR[91,2] = PR[90,2] + 1.358;
   1:L PR[91] R[100]mm/sec CNT100;
   1:  PR[91,1] = PR[90,1] + 35.405;
   1:  PR[91,2] = PR[90,2] + 4.100;
   1:L PR[91] R[100]mm/sec CNT100;
   1:  PR[91,1] = PR[90,1] + 35.024;
   1:  PR[91,2] = PR[90,2] + 5.554;
   1:L PR[91] R[100]mm/sec CNT100;
   1:  PR[91,1] = PR[90,1] + 34.349;
   1:  PR[91,2] = PR[90,2] + 7.037;
   1:L PR[91] R[100]mm/sec CNT100;
   1:  PR[91,1] = PR[90,1] + 33.169;
   1:  PR[91,2] = PR[90,2] + 9.719;
   1:L PR[91] R[100]mm/sec CNT100;
   1:  PR[91,1] = PR[90,1] + 32.346;
   1:  PR[91,2] = PR[90,2] + 10.963;
   1:L PR[91] R[100]mm/sec CNT100;
   1:  PR[91,1] = PR[90,1] + 30.311;
   1:  PR[91,2] = PR[90,2] + 13.494;
   1:L PR[91] R[100]mm/sec CNT100;
   1:  PR[91,1] = PR[90,1] + 29.372;
   1:  PR[91,2] = PR[90,2] + 14.507;
   1:L PR[91] R[100]mm/sec CNT100;
   1:  PR[91,1] = PR[90,1] + 28.356;
   1:  PR[91,2] = PR[90,2] + 15.298;
   1:L PR[91] R[100]mm/sec CNT100;
   1:  PR[91,1] = PR[90,1] + 25.401;
   1:  PR[91,2] = PR[90,2] + 17.446;
   1:L PR[91] R[100]mm/sec CNT100;
   1:  PR[91,1] = PR[90,1] + 24.425;
   1:  PR[91,2] = PR[90,2] + 17.990;
   1:L PR[91] R[100]mm/sec CNT100;
   1:  PR[91,1] = PR[90,1] + 23.397;
   1:  PR[91,2] = PR[90,2] + 18.367;
   1:L PR[91] R[100]mm/sec CNT100;
   1:  PR[91,1] = PR[90,1] + 19.573;
   1:  PR[91,2] = PR[90,2] + 19.864;
   1:L PR[91] R[100]mm/sec CNT100;
   1:  PR[91,1] = PR[90,1] + 18.747;
   1:  PR[91,2] = PR[90,2] + 20.035;
   1:L PR[91] R[100]mm/sec CNT100;
   1:  PR[91,1] = PR[90,1] + 14.166;
   1:  PR[91,2] = PR[90,2] + 20.576;
   1:L PR[91] R[100]mm/sec CNT100;
   1:  PR[91,1] = PR[90,1] + 13.490;
   1:  PR[91,2] = PR[90,2] + 20.611;
   1:L PR[91] R[100]mm/sec CNT100;
   1:  PR[91,1] = PR[90,1] + 12.884;
   1:  PR[91,2] = PR[90,2] + 20.550;
   1:L PR[91] R[100]mm/sec CNT100;
   1:  PR[91,1] = PR[90,1] + 7.918;
   1:  PR[91,2] = PR[90,2] + 19.863;
   1:L PR[91] R[100]mm/sec CNT100;
   1:  PR[91,1] = PR[90,1] + 7.562;
   1:  PR[91,2] = PR[90,2] + 19.771;
   1:L PR[91] R[100]mm/sec CNT100;
   1:  PR[91,1] = PR[90,1] + 2.281;
   1:  PR[91,2] = PR[90,2] + 17.555;
   1:L PR[91] R[100]mm/sec CNT100;
   1:  PR[91,1] = PR[90,1] + 1.628;
   1:  PR[91,2] = PR[90,2] + 17.117;
   1:L PR[91] R[100]mm/sec CNT100;
   1:  PR[91,1] = PR[90,1] + 0.214;
   1:  PR[91,2] = PR[90,2] + 16.533;
   1:L PR[91] R[100]mm/sec CNT100;
   1:  PR[91] = PR[90];
   1:  PR[91,1] = PR[90,1] + -1.083;
   1:  PR[91,2] = PR[90,2] + 17.143;
   1:  PR[91,3] = PR[90,3] + 39.345;
   1:L PR[91] R[100]mm/sec CNT100;
   1:  PR[91,1] = PR[90,1] + -1.525;
   1:  PR[91,2] = PR[90,2] + 17.386;
   1:L PR[91] R[100]mm/sec CNT100;
   1:  PR[91,1] = PR[90,1] + -1.850;
   1:  PR[91,2] = PR[90,2] + 17.604;
   1:L PR[91] R[100]mm/sec CNT100;
   1:  PR[91,1] = PR[90,1] + -1.902;
   1:  PR[91,2] = PR[90,2] + 17.627;
   1:L PR[91] R[100]mm/sec CNT100;
   1:  PR[91,1] = PR[90,1] + -7.214;
   1:  PR[91,2] = PR[90,2] + 19.853;
   1:L PR[91] R[100]mm/sec CNT100;
   1:  PR[91,1] = PR[90,1] + -7.417;
   1:  PR[91,2] = PR[90,2] + 19.905;
   1:L PR[91] R[100]mm/sec CNT100;
   1:  PR[91,1] = PR[90,1] + -7.803;
   1:  PR[91,2] = PR[90,2] + 19.945;
   1:L PR[91] R[100]mm/sec CNT100;
   1:  PR[91,1] = PR[90,1] + -13.139;
   1:  PR[91,2] = PR[90,2] + 20.674;
   1:L PR[91] R[100]mm/sec CNT100;
   1:  PR[91,1] = PR[90,1] + -13.651;
   1:  PR[91,2] = PR[90,2] + 20.647;
   1:L PR[91] R[100]mm/sec CNT100;
   1:  PR[91,1] = PR[90,1] + -18.474;
   1:  PR[91,2] = PR[90,2] + 20.077;
   1:L PR[91] R[100]mm/sec CNT100;
   1:  PR[91,1] = PR[90,1] + -19.180;
   1:  PR[91,2] = PR[90,2] + 19.930;
   1:L PR[91] R[100]mm/sec CNT100;
   1:  PR[91,1] = PR[90,1] + -20.002;
   1:  PR[91,2] = PR[90,2] + 19.625;
   1:L PR[91] R[100]mm/sec CNT100;
   1:  PR[91,1] = PR[90,1] + -24.101;
   1:  PR[91,2] = PR[90,2] + 18.023;
   1:L PR[91] R[100]mm/sec CNT100;
   1:  PR[91,1] = PR[90,1] + -24.948;
   1:  PR[91,2] = PR[90,2] + 17.548;
   1:L PR[91] R[100]mm/sec CNT100;
   1:  PR[91,1] = PR[90,1] + -25.892;
   1:  PR[91,2] = PR[90,2] + 16.813;
   1:L PR[91] R[100]mm/sec CNT100;
   1:  PR[91,1] = PR[90,1] + -29.057;
   1:  PR[91,2] = PR[90,2] + 14.508;
   1:L PR[91] R[100]mm/sec CNT100;
   1:  PR[91,1] = PR[90,1] + -29.878;
   1:  PR[91,2] = PR[90,2] + 13.621;
   1:L PR[91] R[100]mm/sec CNT100;
   1:  PR[91,1] = PR[90,1] + -32.071;
   1:  PR[91,2] = PR[90,2] + 10.898;
   1:L PR[91] R[100]mm/sec CNT100;
   1:  PR[91,1] = PR[90,1] + -32.805;
   1:  PR[91,2] = PR[90,2] + 9.783;
   1:L PR[91] R[100]mm/sec CNT100;
   1:  PR[91,1] = PR[90,1] + -34.698;
   1:  PR[91,2] = PR[90,2] + 5.496;
   1:L PR[91] R[100]mm/sec CNT100;
   1:  PR[91,1] = PR[90,1] + -35.035;
   1:  PR[91,2] = PR[90,2] + 4.194;
   1:L PR[91] R[100]mm/sec CNT100;
   1:  PR[91,1] = PR[90,1] + -35.158;
   1:  PR[91,2] = PR[90,2] + 2.663;
   1:L PR[91] R[100]mm/sec CNT100;
   1:  PR[91,1] = PR[90,1] + -35.576;
   1:  PR[91,2] = PR[90,2] + -0.354;
   1:L PR[91] R[100]mm/sec CNT100;
   1:  PR[91,1] = PR[90,1] + -35.462;
   1:  PR[91,2] = PR[90,2] + -1.791;
   1:L PR[91] R[100]mm/sec CNT100;
   1:  PR[91,1] = PR[90,1] + -35.045;
   1:  PR[91,2] = PR[90,2] + -4.780;
   1:L PR[91] R[100]mm/sec CNT100;
   1:  PR[91,1] = PR[90,1] + -34.698;
   1:  PR[91,2] = PR[90,2] + -6.119;
   1:L PR[91] R[100]mm/sec CNT100;
   1:  PR[91,1] = PR[90,1] + -34.082;
   1:  PR[91,2] = PR[90,2] + -7.494;
   1:L PR[91] R[100]mm/sec CNT100;
   1:  PR[91,1] = PR[90,1] + -32.800;
   1:  PR[91,2] = PR[90,2] + -10.416;
   1:L PR[91] R[100]mm/sec CNT100;
   1:  PR[91,1] = PR[90,1] + -32.067;
   1:  PR[91,2] = PR[90,2] + -11.529;
   1:L PR[91] R[100]mm/sec CNT100;
   1:  PR[91,1] = PR[90,1] + -29.868;
   1:  PR[91,2] = PR[90,2] + -14.255;
   1:L PR[91] R[100]mm/sec CNT100;
   1:  PR[91,1] = PR[90,1] + -29.030;
   1:  PR[91,2] = PR[90,2] + -15.160;
   1:L PR[91] R[100]mm/sec CNT100;
   1:  PR[91,1] = PR[90,1] + -28.114;
   1:  PR[91,2] = PR[90,2] + -15.877;
   1:L PR[91] R[100]mm/sec CNT100;
   1:  PR[91,1] = PR[90,1] + -24.950;
   1:  PR[91,2] = PR[90,2] + -18.170;
   1:L PR[91] R[100]mm/sec CNT100;
   1:  PR[91,1] = PR[90,1] + -24.094;
   1:  PR[91,2] = PR[90,2] + -18.650;
   1:L PR[91] R[100]mm/sec CNT100;
   1:  PR[91,1] = PR[90,1] + -23.193;
   1:  PR[91,2] = PR[90,2] + -18.983;
   1:L PR[91] R[100]mm/sec CNT100;
   1:  PR[91,1] = PR[90,1] + -19.140;
   1:  PR[91,2] = PR[90,2] + -20.564;
   1:L PR[91] R[100]mm/sec CNT100;
   1:  PR[91,1] = PR[90,1] + -18.446;
   1:  PR[91,2] = PR[90,2] + -20.708;
   1:L PR[91] R[100]mm/sec CNT100;
   1:  PR[91,1] = PR[90,1] + -13.612;
   1:  PR[91,2] = PR[90,2] + -21.271;
   1:L PR[91] R[100]mm/sec CNT100;
   1:  PR[91,1] = PR[90,1] + -13.074;
   1:  PR[91,2] = PR[90,2] + -21.299;
   1:L PR[91] R[100]mm/sec CNT100;
   1:  PR[91,1] = PR[90,1] + -12.597;
   1:  PR[91,2] = PR[90,2] + -21.251;
   1:L PR[91] R[100]mm/sec CNT100;
   1:  PR[91,1] = PR[90,1] + -7.393;
   1:  PR[91,2] = PR[90,2] + -20.523;
   1:L PR[91] R[100]mm/sec CNT100;
   1:  PR[91,1] = PR[90,1] + -7.171;
   1:  PR[91,2] = PR[90,2] + -20.465;
   1:L PR[91] R[100]mm/sec CNT100;
   1:  PR[91,1] = PR[90,1] + -1.700;
   1:  PR[91,2] = PR[90,2] + -18.130;
   1:L PR[91] R[100]mm/sec CNT100;
   1:  PR[91,1] = PR[90,1] + -1.403;
   1:  PR[91,2] = PR[90,2] + -17.925;
   1:L PR[91] R[100]mm/sec CNT100;
   1:  PR[91,1] = PR[90,1] + -0.794;
   1:  PR[91,2] = PR[90,2] + -17.746;
   1:L PR[91] R[100]mm/sec CNT100;
   1:  PR[91,1] = PR[90,1] + 0.076;
   1:  PR[91,2] = PR[90,2] + -17.387;
   1:L PR[91] R[100]mm/sec CNT100;
   1:  PR[91,1] = PR[90,1] + 0.986;
   1:  PR[91,2] = PR[90,2] + -17.666;
   1:L PR[91] R[100]mm/sec CNT100;
   1:  PR[91,1] = PR[90,1] + 1.653;
   1:  PR[91,2] = PR[90,2] + -17.997;
   1:L PR[91] R[100]mm/sec CNT100;
   1:  PR[91,1] = PR[90,1] + 1.845;
   1:  PR[91,2] = PR[90,2] + -18.127;
   1:L PR[91] R[100]mm/sec CNT100;
   1:  PR[91,1] = PR[90,1] + 7.324;
   1:  PR[91,2] = PR[90,2] + -20.462;
   1:L PR[91] R[100]mm/sec CNT100;
   1:  PR[91,1] = PR[90,1] + 7.523;
   1:  PR[91,2] = PR[90,2] + -20.514;
   1:L PR[91] R[100]mm/sec CNT100;
   1:  PR[91,1] = PR[90,1] + 7.907;
   1:  PR[91,2] = PR[90,2] + -20.554;
   1:L PR[91] R[100]mm/sec CNT100;
   1:  PR[91,1] = PR[90,1] + 13.255;
   1:  PR[91,2] = PR[90,2] + -21.298;
   1:L PR[91] R[100]mm/sec CNT100;
   1:  PR[91,1] = PR[90,1] + 13.761;
   1:  PR[91,2] = PR[90,2] + -21.271;
   1:L PR[91] R[100]mm/sec CNT100;
   1:  PR[91,1] = PR[90,1] + 18.595;
   1:  PR[91,2] = PR[90,2] + -20.708;
   1:L PR[91] R[100]mm/sec CNT100;
   1:  PR[91,1] = PR[90,1] + 19.300;
   1:  PR[91,2] = PR[90,2] + -20.562;
   1:L PR[91] R[100]mm/sec CNT100;
   1:  PR[91,1] = PR[90,1] + 20.124;
   1:  PR[91,2] = PR[90,2] + -20.258;
   1:L PR[91] R[100]mm/sec CNT100;
   1:  PR[91,1] = PR[90,1] + 24.233;
   1:  PR[91,2] = PR[90,2] + -18.660;
   1:L PR[91] R[100]mm/sec CNT100;
   1:  PR[91,1] = PR[90,1] + 25.076;
   1:  PR[91,2] = PR[90,2] + -18.191;
   1:L PR[91] R[100]mm/sec CNT100;
   1:  PR[91,1] = PR[90,1] + 26.011;
   1:  PR[91,2] = PR[90,2] + -17.466;
   1:L PR[91] R[100]mm/sec CNT100;
   1:  PR[91,1] = PR[90,1] + 29.185;
   1:  PR[91,2] = PR[90,2] + -15.161;
   1:L PR[91] R[100]mm/sec CNT100;
   1:  PR[91,1] = PR[90,1] + 30.007;
   1:  PR[91,2] = PR[90,2] + -14.273;
   1:L PR[91] R[100]mm/sec CNT100;
   1:  PR[91,1] = PR[90,1] + 32.207;
   1:  PR[91,2] = PR[90,2] + -11.541;
   1:L PR[91] R[100]mm/sec CNT100;
   1:  PR[91,1] = PR[90,1] + 32.955;
   1:  PR[91,2] = PR[90,2] + -10.412;
   1:L PR[91] R[100]mm/sec CNT100;
   1:  PR[91,1] = PR[90,1] + 33.573;
   1:  PR[91,2] = PR[90,2] + -9.050;
   1:L PR[91] R[100]mm/sec CNT100;
   1:  PR[91,1] = PR[90,1] + 34.847;
   1:  PR[91,2] = PR[90,2] + -6.162;
   1:L PR[91] R[100]mm/sec CNT100;
   1:  PR[91,1] = PR[90,1] + 35.184;
   1:  PR[91,2] = PR[90,2] + -4.875;
   1:L PR[91] R[100]mm/sec CNT100;
   1:  PR[91,1] = PR[90,1] + 35.314;
   1:  PR[91,2] = PR[90,2] + -3.299;
   1:L PR[91] R[100]mm/sec CNT100;
   1:  PR[91,1] = PR[90,1] + 35.733;
   1:  PR[91,2] = PR[90,2] + -0.271;
   1:L PR[91] R[100]mm/sec CNT100;
   1:  PR[91,1] = PR[90,1] + 35.612;
   1:  PR[91,2] = PR[90,2] + 1.214;
   1:L PR[91] R[100]mm/sec CNT100;
   1:  PR[91,1] = PR[90,1] + 35.196;
   1:  PR[91,2] = PR[90,2] + 4.208;
   1:L PR[91] R[100]mm/sec CNT100;
   1:  PR[91,1] = PR[90,1] + 34.850;
   1:  PR[91,2] = PR[90,2] + 5.526;
   1:L PR[91] R[100]mm/sec CNT100;
   1:  PR[91,1] = PR[90,1] + 34.234;
   1:  PR[91,2] = PR[90,2] + 6.880;
   1:L PR[91] R[100]mm/sec CNT100;
   1:  PR[91,1] = PR[90,1] + 32.955;
   1:  PR[91,2] = PR[90,2] + 9.787;
   1:L PR[91] R[100]mm/sec CNT100;
   1:  PR[91,1] = PR[90,1] + 32.212;
   1:  PR[91,2] = PR[90,2] + 10.910;
   1:L PR[91] R[100]mm/sec CNT100;
   1:  PR[91,1] = PR[90,1] + 30.017;
   1:  PR[91,2] = PR[90,2] + 13.640;
   1:L PR[91] R[100]mm/sec CNT100;
   1:  PR[91,1] = PR[90,1] + 29.178;
   1:  PR[91,2] = PR[90,2] + 14.545;
   1:L PR[91] R[100]mm/sec CNT100;
   1:  PR[91,1] = PR[90,1] + 28.269;
   1:  PR[91,2] = PR[90,2] + 15.253;
   1:L PR[91] R[100]mm/sec CNT100;
   1:  PR[91,1] = PR[90,1] + 25.114;
   1:  PR[91,2] = PR[90,2] + 17.546;
   1:L PR[91] R[100]mm/sec CNT100;
   1:  PR[91,1] = PR[90,1] + 24.264;
   1:  PR[91,2] = PR[90,2] + 18.019;
   1:L PR[91] R[100]mm/sec CNT100;
   1:  PR[91,1] = PR[90,1] + 23.359;
   1:  PR[91,2] = PR[90,2] + 18.352;
   1:L PR[91] R[100]mm/sec CNT100;
   1:  PR[91,1] = PR[90,1] + 19.315;
   1:  PR[91,2] = PR[90,2] + 19.934;
   1:L PR[91] R[100]mm/sec CNT100;
   1:  PR[91,1] = PR[90,1] + 18.622;
   1:  PR[91,2] = PR[90,2] + 20.077;
   1:L PR[91] R[100]mm/sec CNT100;
   1:  PR[91,1] = PR[90,1] + 13.800;
   1:  PR[91,2] = PR[90,2] + 20.648;
   1:L PR[91] R[100]mm/sec CNT100;
   1:  PR[91,1] = PR[90,1] + 13.266;
   1:  PR[91,2] = PR[90,2] + 20.675;
   1:L PR[91] R[100]mm/sec CNT100;
   1:  PR[91,1] = PR[90,1] + 12.787;
   1:  PR[91,2] = PR[90,2] + 20.627;
   1:L PR[91] R[100]mm/sec CNT100;
   1:  PR[91,1] = PR[90,1] + 7.594;
   1:  PR[91,2] = PR[90,2] + 19.909;
   1:L PR[91] R[100]mm/sec CNT100;
   1:  PR[91,1] = PR[90,1] + 7.367;
   1:  PR[91,2] = PR[90,2] + 19.850;
   1:L PR[91] R[100]mm/sec CNT100;
   1:  PR[91,1] = PR[90,1] + 1.993;
   1:  PR[91,2] = PR[90,2] + 17.598;
   1:L PR[91] R[100]mm/sec CNT100;
   1:  PR[91,1] = PR[90,1] + 1.612;
   1:  PR[91,2] = PR[90,2] + 17.343;
   1:L PR[91] R[100]mm/sec CNT100;
   1:  PR[91,1] = PR[90,1] + 0.237;
   1:  PR[91,2] = PR[90,2] + 16.769;
   1:L PR[91] R[100]mm/sec CNT100;
   1:  PR[91] = PR[90];
   1:  PR[91,1] = PR[90,1] + -1.175;
   1:  PR[91,2] = PR[90,2] + 17.411;
   1:  PR[91,3] = PR[90,3] + 39.955;
   1:L PR[91] R[100]mm/sec CNT100;
   1:  PR[91,1] = PR[90,1] + -1.530;
   1:  PR[91,2] = PR[90,2] + 17.631;
   1:L PR[91] R[100]mm/sec CNT100;
   1:  PR[91,1] = PR[90,1] + -7.018;
   1:  PR[91,2] = PR[90,2] + 19.932;
   1:L PR[91] R[100]mm/sec CNT100;
   1:  PR[91,1] = PR[90,1] + -7.113;
   1:  PR[91,2] = PR[90,2] + 19.956;
   1:L PR[91] R[100]mm/sec CNT100;
   1:  PR[91,1] = PR[90,1] + -12.914;
   1:  PR[91,2] = PR[90,2] + 20.738;
   1:L PR[91] R[100]mm/sec CNT100;
   1:  PR[91,1] = PR[90,1] + -13.284;
   1:  PR[91,2] = PR[90,2] + 20.718;
   1:L PR[91] R[100]mm/sec CNT100;
   1:  PR[91,1] = PR[90,1] + -18.349;
   1:  PR[91,2] = PR[90,2] + 20.120;
   1:L PR[91] R[100]mm/sec CNT100;
   1:  PR[91,1] = PR[90,1] + -18.922;
   1:  PR[91,2] = PR[90,2] + 20.001;
   1:L PR[91] R[100]mm/sec CNT100;
   1:  PR[91,1] = PR[90,1] + -19.602;
   1:  PR[91,2] = PR[90,2] + 19.748;
   1:L PR[91] R[100]mm/sec CNT100;
   1:  PR[91,1] = PR[90,1] + -23.939;
   1:  PR[91,2] = PR[90,2] + 18.053;
   1:L PR[91] R[100]mm/sec CNT100;
   1:  PR[91,1] = PR[90,1] + -24.660;
   1:  PR[91,2] = PR[90,2] + 17.649;
   1:L PR[91] R[100]mm/sec CNT100;
   1:  PR[91,1] = PR[90,1] + -25.480;
   1:  PR[91,2] = PR[90,2] + 17.011;
   1:L PR[91] R[100]mm/sec CNT100;
   1:  PR[91,1] = PR[90,1] + -28.861;
   1:  PR[91,2] = PR[90,2] + 14.548;
   1:L PR[91] R[100]mm/sec CNT100;
   1:  PR[91,1] = PR[90,1] + -29.582;
   1:  PR[91,2] = PR[90,2] + 13.769;
   1:L PR[91] R[100]mm/sec CNT100;
   1:  PR[91,1] = PR[90,1] + -31.936;
   1:  PR[91,2] = PR[90,2] + 10.847;
   1:L PR[91] R[100]mm/sec CNT100;
   1:  PR[91,1] = PR[90,1] + -32.590;
   1:  PR[91,2] = PR[90,2] + 9.852;
   1:L PR[91] R[100]mm/sec CNT100;
   1:  PR[91,1] = PR[90,1] + -34.524;
   1:  PR[91,2] = PR[90,2] + 5.470;
   1:L PR[91] R[100]mm/sec CNT100;
   1:  PR[91,1] = PR[90,1] + -34.825;
   1:  PR[91,2] = PR[90,2] + 4.305;
   1:L PR[91] R[100]mm/sec CNT100;
   1:  PR[91,1] = PR[90,1] + -34.936;
   1:  PR[91,2] = PR[90,2] + 2.918;
   1:L PR[91] R[100]mm/sec CNT100;
   1:  PR[91,1] = PR[90,1] + -35.390;
   1:  PR[91,2] = PR[90,2] + -0.354;
   1:L PR[91] R[100]mm/sec CNT100;
   1:  PR[91,1] = PR[90,1] + -35.287;
   1:  PR[91,2] = PR[90,2] + -1.651;
   1:L PR[91] R[100]mm/sec CNT100;
   1:  PR[91,1] = PR[90,1] + -34.835;
   1:  PR[91,2] = PR[90,2] + -4.892;
   1:L PR[91] R[100]mm/sec CNT100;
   1:  PR[91,1] = PR[90,1] + -34.523;
   1:  PR[91,2] = PR[90,2] + -6.094;
   1:L PR[91] R[100]mm/sec CNT100;
   1:  PR[91,1] = PR[90,1] + -33.966;
   1:  PR[91,2] = PR[90,2] + -7.337;
   1:L PR[91] R[100]mm/sec CNT100;
   1:  PR[91,1] = PR[90,1] + -32.585;
   1:  PR[91,2] = PR[90,2] + -10.486;
   1:L PR[91] R[100]mm/sec CNT100;
   1:  PR[91,1] = PR[90,1] + -31.931;
   1:  PR[91,2] = PR[90,2] + -11.478;
   1:L PR[91] R[100]mm/sec CNT100;
   1:  PR[91,1] = PR[90,1] + -29.572;
   1:  PR[91,2] = PR[90,2] + -14.403;
   1:L PR[91] R[100]mm/sec CNT100;
   1:  PR[91,1] = PR[90,1] + -28.833;
   1:  PR[91,2] = PR[90,2] + -15.201;
   1:L PR[91] R[100]mm/sec CNT100;
   1:  PR[91,1] = PR[90,1] + -28.025;
   1:  PR[91,2] = PR[90,2] + -15.834;
   1:L PR[91] R[100]mm/sec CNT100;
   1:  PR[91,1] = PR[90,1] + -24.662;
   1:  PR[91,2] = PR[90,2] + -18.272;
   1:L PR[91] R[100]mm/sec CNT100;
   1:  PR[91,1] = PR[90,1] + -23.931;
   1:  PR[91,2] = PR[90,2] + -18.681;
   1:L PR[91] R[100]mm/sec CNT100;
   1:  PR[91,1] = PR[90,1] + -23.152;
   1:  PR[91,2] = PR[90,2] + -18.969;
   1:L PR[91] R[100]mm/sec CNT100;
   1:  PR[91,1] = PR[90,1] + -18.880;
   1:  PR[91,2] = PR[90,2] + -20.635;
   1:L PR[91] R[100]mm/sec CNT100;
   1:  PR[91,1] = PR[90,1] + -18.320;
   1:  PR[91,2] = PR[90,2] + -20.751;
   1:L PR[91] R[100]mm/sec CNT100;
   1:  PR[91,1] = PR[90,1] + -13.243;
   1:  PR[91,2] = PR[90,2] + -21.342;
   1:L PR[91] R[100]mm/sec CNT100;
   1:  PR[91,1] = PR[90,1] + -12.848;
   1:  PR[91,2] = PR[90,2] + -21.363;
   1:L PR[91] R[100]mm/sec CNT100;
   1:  PR[91,1] = PR[90,1] + -12.498;
   1:  PR[91,2] = PR[90,2] + -21.328;
   1:L PR[91] R[100]mm/sec CNT100;
   1:  PR[91,1] = PR[90,1] + -7.066;
   1:  PR[91,2] = PR[90,2] + -20.567;
   1:L PR[91] R[100]mm/sec CNT100;
   1:  PR[91,1] = PR[90,1] + -6.974;
   1:  PR[91,2] = PR[90,2] + -20.544;
   1:L PR[91] R[100]mm/sec CNT100;
   1:  PR[91,1] = PR[90,1] + -1.723;
   1:  PR[91,2] = PR[90,2] + -18.303;
   1:L PR[91] R[100]mm/sec CNT100;
   1:  PR[91,1] = PR[90,1] + -1.227;
   1:  PR[91,2] = PR[90,2] + -18.103;
   1:L PR[91] R[100]mm/sec CNT100;
   1:  PR[91,1] = PR[90,1] + -0.702;
   1:  PR[91,2] = PR[90,2] + -17.952;
   1:L PR[91] R[100]mm/sec CNT100;
   1:  PR[91,1] = PR[90,1] + 0.096;
   1:  PR[91,2] = PR[90,2] + -17.623;
   1:L PR[91] R[100]mm/sec CNT100;
   1:  PR[91,1] = PR[90,1] + 1.055;
   1:  PR[91,2] = PR[90,2] + -17.917;
   1:L PR[91] R[100]mm/sec CNT100;
   1:  PR[91,1] = PR[90,1] + 1.526;
   1:  PR[91,2] = PR[90,2] + -18.164;
   1:L PR[91] R[100]mm/sec CNT100;
   1:  PR[91,1] = PR[90,1] + 7.126;
   1:  PR[91,2] = PR[90,2] + -20.540;
   1:L PR[91] R[100]mm/sec CNT100;
   1:  PR[91,1] = PR[90,1] + 7.196;
   1:  PR[91,2] = PR[90,2] + -20.559;
   1:L PR[91] R[100]mm/sec CNT100;
   1:  PR[91,1] = PR[90,1] + 7.432;
   1:  PR[91,2] = PR[90,2] + -20.583;
   1:L PR[91] R[100]mm/sec CNT100;
   1:  PR[91,1] = PR[90,1] + 13.029;
   1:  PR[91,2] = PR[90,2] + -21.362;
   1:L PR[91] R[100]mm/sec CNT100;
   1:  PR[91,1] = PR[90,1] + 13.393;
   1:  PR[91,2] = PR[90,2] + -21.343;
   1:L PR[91] R[100]mm/sec CNT100;
   1:  PR[91,1] = PR[90,1] + 18.470;
   1:  PR[91,2] = PR[90,2] + -20.751;
   1:L PR[91] R[100]mm/sec CNT100;
   1:  PR[91,1] = PR[90,1] + 19.041;
   1:  PR[91,2] = PR[90,2] + -20.633;
   1:L PR[91] R[100]mm/sec CNT100;
   1:  PR[91,1] = PR[90,1] + 19.722;
   1:  PR[91,2] = PR[90,2] + -20.382;
   1:L PR[91] R[100]mm/sec CNT100;
   1:  PR[91,1] = PR[90,1] + 24.072;
   1:  PR[91,2] = PR[90,2] + -18.690;
   1:L PR[91] R[100]mm/sec CNT100;
   1:  PR[91,1] = PR[90,1] + 24.789;
   1:  PR[91,2] = PR[90,2] + -18.291;
   1:L PR[91] R[100]mm/sec CNT100;
   1:  PR[91,1] = PR[90,1] + 25.600;
   1:  PR[91,2] = PR[90,2] + -17.662;
   1:L PR[91] R[100]mm/sec CNT100;
   1:  PR[91,1] = PR[90,1] + 28.990;
   1:  PR[91,2] = PR[90,2] + -15.200;
   1:L PR[91] R[100]mm/sec CNT100;
   1:  PR[91,1] = PR[90,1] + 29.712;
   1:  PR[91,2] = PR[90,2] + -14.420;
   1:L PR[91] R[100]mm/sec CNT100;
   1:  PR[91,1] = PR[90,1] + 32.073;
   1:  PR[91,2] = PR[90,2] + -11.489;
   1:L PR[91] R[100]mm/sec CNT100;
   1:  PR[91,1] = PR[90,1] + 32.740;
   1:  PR[91,2] = PR[90,2] + -10.480;
   1:L PR[91] R[100]mm/sec CNT100;
   1:  PR[91,1] = PR[90,1] + 33.295;
   1:  PR[91,2] = PR[90,2] + -9.259;
   1:L PR[91] R[100]mm/sec CNT100;
   1:  PR[91,1] = PR[90,1] + 34.672;
   1:  PR[91,2] = PR[90,2] + -6.135;
   1:L PR[91] R[100]mm/sec CNT100;
   1:  PR[91,1] = PR[90,1] + 34.975;
   1:  PR[91,2] = PR[90,2] + -4.983;
   1:L PR[91] R[100]mm/sec CNT100;
   1:  PR[91,1] = PR[90,1] + 35.092;
   1:  PR[91,2] = PR[90,2] + -3.555;
   1:L PR[91] R[100]mm/sec CNT100;
   1:  PR[91,1] = PR[90,1] + 35.547;
   1:  PR[91,2] = PR[90,2] + -0.271;
   1:L PR[91] R[100]mm/sec CNT100;
   1:  PR[91,1] = PR[90,1] + 35.437;
   1:  PR[91,2] = PR[90,2] + 1.070;
   1:L PR[91] R[100]mm/sec CNT100;
   1:  PR[91,1] = PR[90,1] + 34.986;
   1:  PR[91,2] = PR[90,2] + 4.315;
   1:L PR[91] R[100]mm/sec CNT100;
   1:  PR[91,1] = PR[90,1] + 34.676;
   1:  PR[91,2] = PR[90,2] + 5.499;
   1:L PR[91] R[100]mm/sec CNT100;
   1:  PR[91,1] = PR[90,1] + 34.119;
   1:  PR[91,2] = PR[90,2] + 6.723;
   1:L PR[91] R[100]mm/sec CNT100;
   1:  PR[91,1] = PR[90,1] + 32.741;
   1:  PR[91,2] = PR[90,2] + 9.856;
   1:L PR[91] R[100]mm/sec CNT100;
   1:  PR[91,1] = PR[90,1] + 32.078;
   1:  PR[91,2] = PR[90,2] + 10.857;
   1:L PR[91] R[100]mm/sec CNT100;
   1:  PR[91,1] = PR[90,1] + 29.723;
   1:  PR[91,2] = PR[90,2] + 13.786;
   1:L PR[91] R[100]mm/sec CNT100;
   1:  PR[91,1] = PR[90,1] + 28.984;
   1:  PR[91,2] = PR[90,2] + 14.583;
   1:L PR[91] R[100]mm/sec CNT100;
   1:  PR[91,1] = PR[90,1] + 28.182;
   1:  PR[91,2] = PR[90,2] + 15.208;
   1:L PR[91] R[100]mm/sec CNT100;
   1:  PR[91,1] = PR[90,1] + 24.828;
   1:  PR[91,2] = PR[90,2] + 17.645;
   1:L PR[91] R[100]mm/sec CNT100;
   1:  PR[91,1] = PR[90,1] + 24.103;
   1:  PR[91,2] = PR[90,2] + 18.049;
   1:L PR[91] R[100]mm/sec CNT100;
   1:  PR[91,1] = PR[90,1] + 23.320;
   1:  PR[91,2] = PR[90,2] + 18.337;
   1:L PR[91] R[100]mm/sec CNT100;
   1:  PR[91,1] = PR[90,1] + 19.058;
   1:  PR[91,2] = PR[90,2] + 20.004;
   1:L PR[91] R[100]mm/sec CNT100;
   1:  PR[91,1] = PR[90,1] + 18.498;
   1:  PR[91,2] = PR[90,2] + 20.120;
   1:L PR[91] R[100]mm/sec CNT100;
   1:  PR[91,1] = PR[90,1] + 13.433;
   1:  PR[91,2] = PR[90,2] + 20.719;
   1:L PR[91] R[100]mm/sec CNT100;
   1:  PR[91,1] = PR[90,1] + 13.042;
   1:  PR[91,2] = PR[90,2] + 20.740;
   1:L PR[91] R[100]mm/sec CNT100;
   1:  PR[91,1] = PR[90,1] + 12.690;
   1:  PR[91,2] = PR[90,2] + 20.704;
   1:L PR[91] R[100]mm/sec CNT100;
   1:  PR[91,1] = PR[90,1] + 7.269;
   1:  PR[91,2] = PR[90,2] + 19.954;
   1:L PR[91] R[100]mm/sec CNT100;
   1:  PR[91,1] = PR[90,1] + 7.171;
   1:  PR[91,2] = PR[90,2] + 19.929;
   1:L PR[91] R[100]mm/sec CNT100;
   1:  PR[91,1] = PR[90,1] + 1.706;
   1:  PR[91,2] = PR[90,2] + 17.641;
   1:L PR[91] R[100]mm/sec CNT100;
   1:  PR[91,1] = PR[90,1] + 1.616;
   1:  PR[91,2] = PR[90,2] + 17.580;
   1:L PR[91] R[100]mm/sec CNT100;
   1:  PR[91,1] = PR[90,1] + 1.237;
   1:  PR[91,2] = PR[90,2] + 17.407;
   1:L PR[91] R[100]mm/sec CNT100;
   1:  PR[91,1] = PR[90,1] + 0.248;
   1:  PR[91,2] = PR[90,2] + 17.007;
   1:L PR[91] R[100]mm/sec CNT100;
   1:  PR[91] = PR[90];
   1:  PR[91,1] = PR[90,1] + -1.228;
   1:  PR[91,2] = PR[90,2] + 17.668;
   1:  PR[91,3] = PR[90,3] + 40.565;
   1:L PR[91] R[100]mm/sec CNT100;
   1:  PR[91,1] = PR[90,1] + -1.389;
   1:  PR[91,2] = PR[90,2] + 17.767;
   1:L PR[91] R[100]mm/sec CNT100;
   1:  PR[91,1] = PR[90,1] + -3.118;
   1:  PR[91,2] = PR[90,2] + 18.458;
   1:L PR[91] R[100]mm/sec CNT100;
   1:  PR[91,1] = PR[90,1] + -6.808;
   1:  PR[91,2] = PR[90,2] + 20.004;
   1:L PR[91] R[100]mm/sec CNT100;
   1:  PR[91,1] = PR[90,1] + -12.690;
   1:  PR[91,2] = PR[90,2] + 20.802;
   1:L PR[91] R[100]mm/sec CNT100;
   1:  PR[91,1] = PR[90,1] + -12.917;
   1:  PR[91,2] = PR[90,2] + 20.790;
   1:L PR[91] R[100]mm/sec CNT100;
   1:  PR[91,1] = PR[90,1] + -18.224;
   1:  PR[91,2] = PR[90,2] + 20.163;
   1:L PR[91] R[100]mm/sec CNT100;
   1:  PR[91,1] = PR[90,1] + -18.664;
   1:  PR[91,2] = PR[90,2] + 20.071;
   1:L PR[91] R[100]mm/sec CNT100;
   1:  PR[91,1] = PR[90,1] + -19.201;
   1:  PR[91,2] = PR[90,2] + 19.872;
   1:L PR[91] R[100]mm/sec CNT100;
   1:  PR[91,1] = PR[90,1] + -23.778;
   1:  PR[91,2] = PR[90,2] + 18.083;
   1:L PR[91] R[100]mm/sec CNT100;
   1:  PR[91,1] = PR[90,1] + -24.373;
   1:  PR[91,2] = PR[90,2] + 17.749;
   1:L PR[91] R[100]mm/sec CNT100;
   1:  PR[91,1] = PR[90,1] + -25.068;
   1:  PR[91,2] = PR[90,2] + 17.208;
   1:L PR[91] R[100]mm/sec CNT100;
   1:  PR[91,1] = PR[90,1] + -28.665;
   1:  PR[91,2] = PR[90,2] + 14.588;
   1:L PR[91] R[100]mm/sec CNT100;
   1:  PR[91,1] = PR[90,1] + -29.286;
   1:  PR[91,2] = PR[90,2] + 13.917;
   1:L PR[91] R[100]mm/sec CNT100;
   1:  PR[91,1] = PR[90,1] + -31.800;
   1:  PR[91,2] = PR[90,2] + 10.796;
   1:L PR[91] R[100]mm/sec CNT100;
   1:  PR[91,1] = PR[90,1] + -32.375;
   1:  PR[91,2] = PR[90,2] + 9.922;
   1:L PR[91] R[100]mm/sec CNT100;
   1:  PR[91,1] = PR[90,1] + -34.349;
   1:  PR[91,2] = PR[90,2] + 5.445;
   1:L PR[91] R[100]mm/sec CNT100;
   1:  PR[91,1] = PR[90,1] + -34.615;
   1:  PR[91,2] = PR[90,2] + 4.416;
   1:L PR[91] R[100]mm/sec CNT100;
   1:  PR[91,1] = PR[90,1] + -34.715;
   1:  PR[91,2] = PR[90,2] + 3.173;
   1:L PR[91] R[100]mm/sec CNT100;
   1:  PR[91,1] = PR[90,1] + -35.204;
   1:  PR[91,2] = PR[90,2] + -0.354;
   1:L PR[91] R[100]mm/sec CNT100;
   1:  PR[91,1] = PR[90,1] + -35.112;
   1:  PR[91,2] = PR[90,2] + -1.511;
   1:L PR[91] R[100]mm/sec CNT100;
   1:  PR[91,1] = PR[90,1] + -34.625;
   1:  PR[91,2] = PR[90,2] + -5.003;
   1:L PR[91] R[100]mm/sec CNT100;
   1:  PR[91,1] = PR[90,1] + -34.349;
   1:  PR[91,2] = PR[90,2] + -6.069;
   1:L PR[91] R[100]mm/sec CNT100;
   1:  PR[91,1] = PR[90,1] + -33.850;
   1:  PR[91,2] = PR[90,2] + -7.180;
   1:L PR[91] R[100]mm/sec CNT100;
   1:  PR[91,1] = PR[90,1] + -32.369;
   1:  PR[91,2] = PR[90,2] + -10.555;
   1:L PR[91] R[100]mm/sec CNT100;
   1:  PR[91,1] = PR[90,1] + -31.795;
   1:  PR[91,2] = PR[90,2] + -11.428;
   1:L PR[91] R[100]mm/sec CNT100;
   1:  PR[91,1] = PR[90,1] + -29.275;
   1:  PR[91,2] = PR[90,2] + -14.552;
   1:L PR[91] R[100]mm/sec CNT100;
   1:  PR[91,1] = PR[90,1] + -28.636;
   1:  PR[91,2] = PR[90,2] + -15.242;
   1:L PR[91] R[100]mm/sec CNT100;
   1:  PR[91,1] = PR[90,1] + -27.936;
   1:  PR[91,2] = PR[90,2] + -15.790;
   1:L PR[91] R[100]mm/sec CNT100;
   1:  PR[91,1] = PR[90,1] + -24.373;
   1:  PR[91,2] = PR[90,2] + -18.373;
   1:L PR[91] R[100]mm/sec CNT100;
   1:  PR[91,1] = PR[90,1] + -23.769;
   1:  PR[91,2] = PR[90,2] + -18.711;
   1:L PR[91] R[100]mm/sec CNT100;
   1:  PR[91,1] = PR[90,1] + -23.112;
   1:  PR[91,2] = PR[90,2] + -18.954;
   1:L PR[91] R[100]mm/sec CNT100;
   1:  PR[91,1] = PR[90,1] + -18.620;
   1:  PR[91,2] = PR[90,2] + -20.706;
   1:L PR[91] R[100]mm/sec CNT100;
   1:  PR[91,1] = PR[90,1] + -18.194;
   1:  PR[91,2] = PR[90,2] + -20.794;
   1:L PR[91] R[100]mm/sec CNT100;
   1:  PR[91,1] = PR[90,1] + -12.873;
   1:  PR[91,2] = PR[90,2] + -21.414;
   1:L PR[91] R[100]mm/sec CNT100;
   1:  PR[91,1] = PR[90,1] + -12.622;
   1:  PR[91,2] = PR[90,2] + -21.427;
   1:L PR[91] R[100]mm/sec CNT100;
   1:  PR[91,1] = PR[90,1] + -12.399;
   1:  PR[91,2] = PR[90,2] + -21.404;
   1:L PR[91] R[100]mm/sec CNT100;
   1:  PR[91,1] = PR[90,1] + -6.761;
   1:  PR[91,2] = PR[90,2] + -20.615;
   1:L PR[91] R[100]mm/sec CNT100;
   1:  PR[91,1] = PR[90,1] + -4.016;
   1:  PR[91,2] = PR[90,2] + -19.444;
   1:L PR[91] R[100]mm/sec CNT100;
   1:  PR[91,1] = PR[90,1] + -1.135;
   1:  PR[91,2] = PR[90,2] + -18.283;
   1:L PR[91] R[100]mm/sec CNT100;
   1:  PR[91,1] = PR[90,1] + -0.880;
   1:  PR[91,2] = PR[90,2] + -18.239;
   1:L PR[91] R[100]mm/sec CNT100;
   1:  PR[91,1] = PR[90,1] + -0.618;
   1:  PR[91,2] = PR[90,2] + -18.162;
   1:L PR[91] R[100]mm/sec CNT100;
   1:  PR[91,1] = PR[90,1] + 0.116;
   1:  PR[91,2] = PR[90,2] + -17.860;
   1:L PR[91] R[100]mm/sec CNT100;
   1:  PR[91,1] = PR[90,1] + 1.110;
   1:  PR[91,2] = PR[90,2] + -18.164;
   1:L PR[91] R[100]mm/sec CNT100;
   1:  PR[91,1] = PR[90,1] + 1.497;
   1:  PR[91,2] = PR[90,2] + -18.367;
   1:L PR[91] R[100]mm/sec CNT100;
   1:  PR[91,1] = PR[90,1] + 4.169;
   1:  PR[91,2] = PR[90,2] + -19.443;
   1:L PR[91] R[100]mm/sec CNT100;
   1:  PR[91,1] = PR[90,1] + 6.913;
   1:  PR[91,2] = PR[90,2] + -20.612;
   1:L PR[91] R[100]mm/sec CNT100;
   1:  PR[91,1] = PR[90,1] + 12.803;
